C09140=1188.823,174.713,-56.680,-178.031,6.459,148.597
C09141=1188.828,174.463,-56.658,-178.034,6.458,148.598
C09142=1188.832,174.215,-56.637,-178.036,6.457,148.598
C09143=1188.837,173.966,-56.613,-178.039,6.455,148.599
C09144=1188.841,173.716,-56.591,-178.041,6.453,148.599
C09145=1188.846,173.468,-56.569,-178.044,6.451,148.599
C09146=1188.851,173.219,-56.546,-178.047,6.450,148.600
C09147=1188.856,172.970,-56.524,-178.049,6.448,148.600
C09148=1188.860,172.721,-56.502,-178.052,6.446,148.600
C09149=1188.865,172.472,-56.479,-178.055,6.444,148.601
C09150=1188.870,172.223,-56.457,-178.057,6.442,148.601
C09151=1188.874,171.974,-56.435,-178.060,6.441,148.601
C09152=1188.879,171.725,-56.412,-178.063,6.439,148.602
C09153=1188.884,171.476,-56.390,-178.065,6.437,148.602
C09154=1188.888,171.228,-56.369,-178.068,6.435,148.603
C09155=1188.893,170.978,-56.347,-178.071,6.433,148.603
C09156=1188.898,170.729,-56.324,-178.073,6.432,148.603
C09157=1188.902,170.480,-56.301,-178.076,6.430,148.604
C09158=1188.907,170.231,-56.279,-178.079,6.428,148.604
C09159=1188.911,169.983,-56.258,-178.081,6.426,148.604
C09160=1188.916,169.733,-56.235,-178.084,6.425,148.605
C09161=1188.921,169.484,-56.213,-178.087,6.423,148.605
C09162=1188.925,169.235,-56.191,-178.089,6.422,148.605
C09163=1188.930,168.987,-56.169,-178.092,6.420,148.606
C09164=1188.935,168.737,-56.146,-178.095,6.419,148.606
C09165=1188.940,168.489,-56.125,-178.097,6.417,148.607
C09166=1188.944,168.239,-56.103,-178.100,6.415,148.607
C09167=1188.949,167.991,-56.081,-178.103,6.413,148.608
C09168=1188.953,167.741,-56.059,-178.105,6.411,148.608
C09169=1188.958,167.493,-56.037,-178.108,6.410,148.608
C09170=1188.963,167.243,-56.015,-178.111,6.408,148.609
C09171=1188.968,166.994,-55.993,-178.114,6.406,148.609
C09172=1188.972,166.745,-55.971,-178.116,6.404,148.609
C09173=1188.977,166.496,-55.949,-178.119,6.403,148.610
C09174=1188.982,166.247,-55.927,-178.122,6.401,148.610
C09175=1188.986,165.998,-55.905,-178.124,6.400,148.610
C09176=1188.991,165.750,-55.884,-178.126,6.398,148.611
C09177=1188.996,165.500,-55.862,-178.129,6.396,148.611
C09178=1189.001,165.251,-55.839,-178.132,6.394,148.612
C09179=1189.005,165.002,-55.817,-178.134,6.393,148.612
C09180=1189.010,164.753,-55.796,-178.137,6.391,148.612
C09181=1189.015,164.504,-55.774,-178.140,6.389,148.613
C09182=1189.019,164.255,-55.752,-178.142,6.387,148.613
C09183=1189.024,164.006,-55.730,-178.146,6.386,148.614
C09184=1189.029,163.757,-55.708,-178.148,6.384,148.614
C09185=1189.033,163.509,-55.687,-178.151,6.382,148.614
C09186=1189.038,163.259,-55.664,-178.153,6.381,148.615
C09187=1189.043,163.011,-55.643,-178.156,6.380,148.615
C09188=1189.047,162.762,-55.621,-178.158,6.378,148.616
C09189=1189.052,162.512,-55.600,-178.161,6.376,148.616
C09190=1189.057,162.264,-55.578,-178.164,6.374,148.616
C09191=1189.061,162.014,-55.556,-178.166,6.372,148.617
C09192=1189.066,161.766,-55.534,-178.169,6.371,148.617
C09193=1189.070,161.516,-55.512,-178.172,6.369,148.617
C09194=1189.075,161.268,-55.491,-178.174,6.368,148.618
C09195=1189.080,161.018,-55.470,-178.177,6.366,148.618
C09196=1189.085,160.769,-55.448,-178.180,6.365,148.619
C09197=1189.089,160.520,-55.426,-178.182,6.363,148.619
C09198=1189.094,160.272,-55.404,-178.185,6.361,148.619
C09199=1189.099,160.022,-55.383,-178.188,6.359,148.620
C09200=1189.104,159.773,-55.361,-178.190,6.358,148.620
C09201=1189.109,159.525,-55.340,-178.193,6.356,148.621
C09202=1189.112,159.276,-55.318,-178.195,6.355,148.621
C09203=1189.118,159.006,-55.295,-178.198,6.352,148.621
C09204=1189.123,158.737,-55.271,-178.202,6.351,148.622
C09205=1189.128,158.468,-55.248,-178.204,6.349,148.622
C09206=1189.132,158.199,-55.225,-178.207,6.347,148.623
C09207=1189.138,157.950,-55.204,-178.210,6.346,148.623
C09208=1189.142,157.701,-55.182,-178.212,6.344,148.623
C09209=1189.147,157.453,-55.161,-178.215,6.343,148.624
C09210=1189.152,157.203,-55.139,-178.218,6.341,148.624
C09211=1189.157,156.954,-55.118,-178.220,6.340,148.625
C09212=1189.162,156.706,-55.096,-178.223,6.338,148.625
C09213=1189.166,156.456,-55.075,-178.226,6.336,148.626
C09214=1189.170,156.207,-55.054,-178.228,6.334,148.626
C09215=1189.175,155.958,-55.033,-178.230,6.333,148.626
C09216=1189.180,155.709,-55.011,-178.233,6.332,148.627
C09217=1189.185,155.459,-54.990,-178.236,6.330,148.627
C09218=1189.190,155.211,-54.968,-178.239,6.328,148.628
C09219=1189.194,154.962,-54.947,-178.242,6.327,148.628
C09220=1189.199,154.713,-54.926,-178.244,6.325,148.628
C09221=1189.203,154.464,-54.904,-178.247,6.323,148.629
C09222=1189.209,154.215,-54.883,-178.249,6.322,148.629
C09223=1189.213,153.966,-54.861,-178.252,6.320,148.630
C09224=1189.218,153.717,-54.841,-178.255,6.319,148.630
C09225=1189.222,153.468,-54.819,-178.258,6.317,148.631
C09226=1189.227,153.218,-54.798,-178.260,6.315,148.631
C09227=1189.232,152.969,-54.777,-178.262,6.314,148.631
C09228=1189.237,152.721,-54.756,-178.265,6.313,148.632
C09229=1189.241,152.471,-54.734,-178.268,6.311,148.632
C09230=1189.246,152.222,-54.713,-178.271,6.309,148.632
C09231=1189.250,151.973,-54.692,-178.273,6.307,148.633
C09232=1189.256,151.724,-54.671,-178.276,6.306,148.633
C09233=1189.260,151.475,-54.650,-178.278,6.305,148.634
C09234=1189.266,151.226,-54.629,-178.281,6.303,148.634
C09235=1189.269,150.977,-54.607,-178.284,6.301,148.635
C09236=1189.274,150.728,-54.586,-178.287,6.300,148.635
C09237=1189.280,150.478,-54.565,-178.289,6.298,148.635
C09238=1189.284,150.230,-54.544,-178.292,6.297,148.636
C09239=1189.289,149.981,-54.523,-178.294,6.295,148.636
C09240=1189.293,149.732,-54.503,-178.297,6.294,148.637
C09241=1189.298,149.483,-54.481,-178.300,6.292,148.637
C09242=1189.303,149.233,-54.460,-178.303,6.290,148.637
C09243=1189.307,148.984,-54.440,-178.305,6.289,148.638
C09244=1189.312,148.735,-54.419,-178.308,6.288,148.638
C09245=1189.317,148.487,-54.397,-178.311,6.286,148.639
C09246=1189.322,148.238,-54.377,-178.313,6.284,148.639
C09247=1189.327,147.988,-54.356,-178.316,6.282,148.640
C09248=1189.331,147.739,-54.335,-178.318,6.281,148.640
C09249=1189.336,147.490,-54.313,-178.321,6.280,148.640
C09250=1189.341,147.241,-54.292,-178.324,6.278,148.641
C09251=1189.345,146.992,-54.272,-178.327,6.277,148.641
C09252=1189.350,146.743,-54.251,-178.329,6.275,148.642
C09253=1189.355,146.494,-54.231,-178.331,6.274,148.642
C09254=1189.360,146.245,-54.209,-178.334,6.272,148.643
C09255=1189.364,145.996,-54.188,-178.337,6.270,148.643
C09256=1189.369,145.747,-54.168,-178.340,6.269,148.643
C09257=1189.373,145.497,-54.147,-178.342,6.268,148.644
C09258=1189.378,145.248,-54.126,-178.345,6.266,148.644
C09259=1189.383,144.999,-54.105,-178.347,6.264,148.645
C09260=1189.388,144.750,-54.084,-178.350,6.263,148.645
C09261=1189.392,144.501,-54.064,-178.353,6.261,148.646
C09262=1189.397,144.251,-54.043,-178.355,6.260,148.646
C09263=1189.402,144.003,-54.022,-178.358,6.258,148.646
C09264=1189.407,143.754,-54.001,-178.361,6.257,148.647
C09265=1189.411,143.505,-53.981,-178.363,6.255,148.647
C09266=1189.416,143.256,-53.960,-178.366,6.254,148.648
C09267=1189.421,143.007,-53.939,-178.369,6.253,148.648
C09268=1189.426,142.757,-53.918,-178.371,6.251,148.649
C09269=1189.430,142.508,-53.898,-178.374,6.249,148.649
C09270=1189.435,142.260,-53.878,-178.376,6.248,148.649
C09271=1189.440,142.010,-53.857,-178.379,6.247,148.650
C09272=1189.444,141.761,-53.836,-178.382,6.245,148.650
C09273=1189.450,141.512,-53.815,-178.385,6.243,148.651
C09274=1189.454,141.263,-53.795,-178.387,6.242,148.651
C09275=1189.459,141.014,-53.775,-178.390,6.241,148.652
C09276=1189.464,140.764,-53.754,-178.393,6.239,148.652
C09277=1189.468,140.515,-53.734,-178.395,6.237,148.653
C09278=1189.474,140.266,-53.713,-178.398,6.236,148.653
C09279=1189.478,140.017,-53.693,-178.400,6.235,148.653
C09280=1189.482,139.768,-53.672,-178.403,6.233,148.654
C09281=1189.488,139.519,-53.651,-178.405,6.232,148.654
C09282=1189.492,139.270,-53.631,-178.408,6.230,148.655
C09283=1189.497,139.021,-53.611,-178.411,6.229,148.655
C09284=1189.502,138.772,-53.590,-178.414,6.227,148.656
C09285=1189.506,138.522,-53.570,-178.416,6.226,148.656
C09286=1189.511,138.273,-53.550,-178.419,6.225,148.656
C09287=1189.516,138.024,-53.529,-178.422,6.223,148.657
C09288=1189.521,137.775,-53.508,-178.425,6.221,148.657
C09289=1189.525,137.526,-53.488,-178.427,6.220,148.658
C09290=1189.530,137.277,-53.468,-178.430,6.219,148.658
C09291=1189.535,137.027,-53.447,-178.432,6.217,148.659
C09292=1189.539,136.778,-53.427,-178.434,6.216,148.659
C09293=1189.544,136.529,-53.406,-178.438,6.215,148.660
C09294=1189.548,136.280,-53.386,-178.440,6.213,148.660
C09295=1189.554,136.031,-53.366,-178.443,6.211,148.660
C09296=1189.559,135.782,-53.346,-178.445,6.210,148.661
C09297=1189.563,135.533,-53.325,-178.448,6.209,148.661
C09298=1189.568,135.284,-53.306,-178.451,6.207,148.662
C09299=1189.573,135.034,-53.285,-178.453,6.206,148.662
C09300=1189.577,134.786,-53.264,-178.456,6.204,148.663
C09301=1189.582,134.536,-53.245,-178.459,6.203,148.663
C09302=1189.587,134.287,-53.224,-178.462,6.201,148.664
C09303=1189.592,134.038,-53.203,-178.464,6.200,148.664
C09304=1189.597,133.788,-53.184,-178.467,6.199,148.665
C09305=1189.602,133.540,-53.164,-178.470,6.197,148.665
C09306=1189.606,133.291,-53.143,-178.472,6.196,148.665
C09307=1189.612,133.022,-53.122,-178.475,6.195,148.666
C09308=1189.616,132.754,-53.100,-178.478,6.193,148.666
C09309=1189.622,132.485,-53.078,-178.480,6.191,148.667
C09310=1189.627,132.216,-53.057,-178.483,6.190,148.667
C09311=1189.631,131.967,-53.037,-178.486,6.188,148.668
C09312=1189.636,131.718,-53.017,-178.488,6.187,148.668
C09313=1189.641,131.469,-52.996,-178.491,6.186,148.669
C09314=1189.646,131.219,-52.977,-178.494,6.184,148.669
C09315=1189.650,130.970,-52.956,-178.496,6.183,148.670
C09316=1189.655,130.722,-52.936,-178.499,6.181,148.670
C09317=1189.660,130.472,-52.917,-178.502,6.180,148.671
C09318=1189.665,130.223,-52.896,-178.504,6.179,148.671
C09319=1189.669,129.974,-52.876,-178.507,6.177,148.671
C09320=1189.674,129.724,-52.857,-178.510,6.176,148.672
C09321=1189.679,129.476,-52.837,-178.512,6.175,148.672
C09322=1189.684,129.226,-52.817,-178.515,6.173,148.673
C09323=1189.688,128.977,-52.797,-178.518,6.171,148.673
C09324=1189.693,128.728,-52.777,-178.520,6.171,148.674
C09325=1189.698,128.479,-52.756,-178.523,6.169,148.674
C09326=1189.704,128.230,-52.737,-178.526,6.167,148.675
C09327=1189.708,127.981,-52.717,-178.528,6.166,148.675
C09328=1189.713,127.731,-52.697,-178.531,6.165,148.676
C09329=1189.718,127.482,-52.677,-178.534,6.163,148.676
C09330=1189.723,127.233,-52.657,-178.536,6.162,148.677
C09331=1189.727,126.984,-52.638,-178.539,6.161,148.677
C09332=1189.732,126.734,-52.618,-178.542,6.159,148.678
C09333=1189.736,126.485,-52.598,-178.544,6.158,148.678
C09334=1189.742,126.236,-52.578,-178.547,6.156,148.679
C09335=1189.746,125.987,-52.559,-178.550,6.155,148.679
C09336=1189.750,125.738,-52.539,-178.552,6.154,148.679
C09337=1189.755,125.489,-52.519,-178.555,6.152,148.680
C09338=1189.760,125.240,-52.500,-178.557,6.151,148.680
C09339=1189.765,124.991,-52.479,-178.560,6.150,148.681
C09340=1189.770,124.741,-52.460,-178.563,6.148,148.681
C09341=1189.775,124.492,-52.441,-178.565,6.147,148.682
C09342=1189.780,124.243,-52.421,-178.568,6.146,148.682
C09343=1189.784,123.994,-52.401,-178.571,6.144,148.683
C09344=1189.789,123.744,-52.381,-178.573,6.143,148.683
C09345=1189.794,123.495,-52.362,-178.576,6.141,148.684
C09346=1189.799,123.246,-52.342,-178.578,6.141,148.684
C09347=1189.803,122.997,-52.322,-178.581,6.139,148.685
C09348=1189.808,122.748,-52.303,-178.584,6.137,148.685
C09349=1189.813,122.499,-52.283,-178.586,6.137,148.686
C09350=1189.817,122.249,-52.264,-178.589,6.135,148.686
C09351=1189.823,122.000,-52.244,-178.592,6.133,148.686
C09352=1189.828,121.751,-52.225,-178.594,6.133,148.687
C09353=1189.832,121.502,-52.204,-178.597,6.131,148.687
C09354=1189.837,121.253,-52.185,-178.599,6.130,148.688
C09355=1189.841,121.004,-52.166,-178.602,6.129,148.689
C09356=1189.846,120.754,-52.146,-178.605,6.127,148.689
C09357=1189.851,120.505,-52.127,-178.607,6.126,148.689
C09358=1189.856,120.256,-52.107,-178.610,6.125,148.690
C09359=1189.861,120.007,-52.088,-178.612,6.124,148.690
C09360=1189.865,119.758,-52.069,-178.615,6.122,148.691
C09361=1189.870,119.508,-52.049,-178.618,6.120,148.691
C09362=1189.876,119.259,-52.030,-178.620,6.120,148.692
C09363=1189.880,119.010,-52.010,-178.623,6.118,148.692
C09364=1189.885,118.761,-51.990,-178.626,6.117,148.693
C09365=1189.889,118.512,-51.971,-178.628,6.115,148.693
C09366=1189.894,118.263,-51.952,-178.631,6.114,148.694
C09367=1189.899,118.014,-51.932,-178.634,6.113,148.694
C09368=1189.904,117.764,-51.913,-178.636,6.111,148.695
C09369=1189.909,117.516,-51.894,-178.639,6.110,148.695
C09370=1189.914,117.265,-51.875,-178.642,6.109,148.696
C09371=1189.919,117.016,-51.855,-178.644,6.107,148.696
C09372=1189.924,116.767,-51.836,-178.647,6.107,148.697
C09373=1189.928,116.518,-51.817,-178.650,6.105,148.697
C09374=1189.933,116.269,-51.798,-178.652,6.104,148.698
C09375=1189.938,116.019,-51.778,-178.655,6.103,148.698
C09376=1189.943,115.771,-51.759,-178.658,6.101,148.699
C09377=1189.947,115.521,-51.740,-178.660,6.100,148.699
C09378=1189.952,115.272,-51.720,-178.663,6.099,148.700
C09379=1189.957,115.023,-51.701,-178.665,6.098,148.700
C09380=1189.961,114.773,-51.682,-178.668,6.096,148.700
C09381=1189.967,114.525,-51.662,-178.671,6.095,148.701
C09382=1189.971,114.275,-51.644,-178.673,6.094,148.701
C09383=1189.976,114.026,-51.625,-178.676,6.092,148.702
C09384=1189.981,113.776,-51.605,-178.679,6.091,148.703
C09385=1189.986,113.528,-51.586,-178.681,6.090,148.703
C09386=1189.991,113.278,-51.567,-178.684,6.089,148.704
C09387=1189.995,113.029,-51.549,-178.687,6.087,148.704
C09388=1190.000,112.779,-51.529,-178.689,6.087,148.705
C09389=1190.006,112.531,-51.510,-178.692,6.085,148.705
C09390=1190.010,112.281,-51.491,-178.694,6.084,148.705
C09391=1190.015,112.032,-51.471,-178.697,6.083,148.706
C09392=1190.019,111.783,-51.453,-178.700,6.081,148.706
C09393=1190.025,111.534,-51.434,-178.702,6.080,148.707
C09394=1190.029,111.284,-51.414,-178.705,6.078,148.707
C09395=1190.034,111.036,-51.395,-178.707,6.078,148.708
C09396=1190.039,110.785,-51.377,-178.711,6.076,148.709
C09397=1190.044,110.537,-51.358,-178.713,6.075,148.709
C09398=1190.049,110.288,-51.339,-178.715,6.074,148.709
C09399=1190.053,110.038,-51.320,-178.718,6.073,148.710
C09400=1190.059,109.789,-51.301,-178.721,6.071,148.710
C09401=1190.063,109.540,-51.282,-178.723,6.071,148.711
C09402=1190.068,109.290,-51.263,-178.726,6.069,148.711
C09403=1190.072,109.041,-51.244,-178.729,6.067,148.712
C09404=1190.078,108.792,-51.225,-178.731,6.067,148.712
C09405=1190.082,108.542,-51.207,-178.734,6.065,148.713
C09406=1190.087,108.294,-51.187,-178.737,6.064,148.714
C09407=1190.092,108.044,-51.169,-178.739,6.062,148.714
C09408=1190.097,107.795,-51.150,-178.742,6.062,148.714
C09409=1190.101,107.546,-51.131,-178.745,6.060,148.715
C09410=1190.107,107.296,-51.112,-178.747,6.059,148.715
C09411=1190.111,107.028,-51.092,-178.750,6.058,148.716
C09412=1190.117,106.760,-51.072,-178.753,6.056,148.716
C09413=1190.122,106.491,-51.051,-178.755,6.056,148.717
C09414=1190.127,106.223,-51.031,-178.759,6.054,148.718
C09415=1190.132,105.974,-51.012,-178.761,6.052,148.718
C09416=1190.137,105.724,-50.994,-178.764,6.052,148.719
C09417=1190.141,105.476,-50.975,-178.767,6.050,148.719
C09418=1190.147,105.226,-50.956,-178.769,6.049,148.720
C09419=1190.151,104.977,-50.937,-178.772,6.048,148.720
C09420=1190.157,104.727,-50.919,-178.774,6.047,148.721
C09421=1190.161,104.478,-50.900,-178.777,6.046,148.721
C09422=1190.166,104.229,-50.882,-178.779,6.045,148.722
C09423=1190.171,103.980,-50.863,-178.782,6.043,148.722
C09424=1190.175,103.730,-50.844,-178.785,6.042,148.723
C09425=1190.180,103.481,-50.826,-178.787,6.041,148.723
C09426=1190.186,103.232,-50.807,-178.790,6.040,148.724
C09427=1190.190,102.982,-50.789,-178.793,6.038,148.724
C09428=1190.195,102.733,-50.770,-178.795,6.038,148.725
C09429=1190.200,102.484,-50.751,-178.798,6.036,148.725
C09430=1190.204,102.234,-50.733,-178.801,6.035,148.726
C09431=1190.209,101.986,-50.714,-178.803,6.034,148.726
C09432=1190.215,101.736,-50.696,-178.805,6.033,148.727
C09433=1190.220,101.487,-50.678,-178.809,6.031,148.727
C09434=1190.224,101.238,-50.659,-178.811,6.030,148.728
C09435=1190.229,100.988,-50.640,-178.814,6.029,148.728
C09436=1190.234,100.739,-50.622,-178.816,6.028,148.729
C09437=1190.238,100.490,-50.603,-178.819,6.027,148.729
C09438=1190.243,100.241,-50.585,-178.821,6.026,148.730
C09439=1190.249,99.991,-50.566,-178.825,6.024,148.731
C09440=1190.254,99.742,-50.548,-178.827,6.023,148.731
C09441=1190.258,99.493,-50.529,-178.829,6.023,148.731
C09442=1190.263,99.244,-50.511,-178.832,6.021,148.732
C09443=1190.268,98.994,-50.493,-178.834,6.020,148.732
C09444=1190.272,98.745,-50.474,-178.837,6.019,148.733
C09445=1190.277,98.496,-50.456,-178.840,6.018,148.733
C09446=1190.282,98.247,-50.438,-178.843,6.017,148.734
C09447=1190.288,97.997,-50.419,-178.845,6.016,148.735
C09448=1190.292,97.747,-50.401,-178.848,6.014,148.735
C09449=1190.297,97.499,-50.382,-178.850,6.013,148.736
C09450=1190.301,97.250,-50.364,-178.853,6.012,148.736
C09451=1190.306,97.000,-50.346,-178.856,6.011,148.737
C09452=1190.312,96.751,-50.328,-178.859,6.010,148.737
C09453=1190.316,96.501,-50.309,-178.861,6.009,148.738
C09454=1190.321,96.252,-50.291,-178.864,6.007,148.738
C09455=1190.326,96.003,-50.273,-178.866,6.006,148.739
C09456=1190.331,95.754,-50.255,-178.868,6.006,148.739
C09457=1190.336,95.505,-50.237,-178.872,6.004,148.740
C09458=1190.340,95.255,-50.218,-178.874,6.003,148.740
C09459=1190.346,95.006,-50.200,-178.877,6.002,148.741
C09460=1190.351,94.756,-50.182,-178.879,6.001,148.741
C09461=1190.355,94.507,-50.164,-178.882,6.000,148.742
C09462=1190.360,94.258,-50.146,-178.884,5.999,148.742
C09463=1190.365,94.008,-50.128,-178.888,5.997,148.743
C09464=1190.370,93.759,-50.110,-178.890,5.996,148.743
C09465=1190.375,93.510,-50.092,-178.892,5.996,148.744
C09466=1190.379,93.261,-50.074,-178.895,5.994,148.744
C09467=1190.384,93.011,-50.056,-178.898,5.994,148.745
C09468=1190.389,92.762,-50.038,-178.900,5.992,148.746
C09469=1190.394,92.512,-50.019,-178.903,5.991,148.746
C09470=1190.399,92.263,-50.001,-178.906,5.990,148.747
C09471=1190.404,92.014,-49.983,-178.908,5.989,148.747
C09472=1190.409,91.765,-49.965,-178.910,5.988,148.748
C09473=1190.414,91.515,-49.947,-178.914,5.987,148.748
C09474=1190.419,91.266,-49.929,-178.916,5.986,148.749
C09475=1190.424,91.017,-49.911,-178.919,5.984,148.749
C09476=1190.429,90.768,-49.893,-178.921,5.983,148.750
C09477=1190.433,90.518,-49.874,-178.924,5.982,148.750
C09478=1190.438,90.269,-49.856,-178.926,5.981,148.751
C09479=1190.443,90.020,-49.838,-178.929,5.981,148.752
C09480=1190.448,89.770,-49.821,-178.932,5.979,148.752
C09481=1190.453,89.521,-49.803,-178.934,5.978,148.753
C09482=1190.458,89.272,-49.785,-178.937,5.977,148.753
C09483=1190.463,89.022,-49.767,-178.940,5.976,148.754
C09484=1190.468,88.773,-49.749,-178.942,5.975,148.754
C09485=1190.473,88.524,-49.731,-178.945,5.974,148.755
C09486=1190.478,88.275,-49.713,-178.947,5.973,148.755
C09487=1190.481,88.025,-49.696,-178.950,5.971,148.756
C09488=1190.486,87.776,-49.678,-178.953,5.971,148.756
C09489=1190.491,87.526,-49.660,-178.955,5.970,148.757
C09490=1190.496,87.277,-49.642,-178.958,5.968,148.757
C09491=1190.501,87.028,-49.624,-178.960,5.968,148.758
C09492=1190.506,86.779,-49.606,-178.963,5.966,148.758
C09493=1190.511,86.530,-49.588,-178.966,5.965,148.759
C09494=1190.516,86.280,-49.571,-178.968,5.965,148.759
C09495=1190.521,86.031,-49.553,-178.971,5.963,148.760
C09496=1190.526,85.781,-49.535,-178.973,5.962,148.761
C09497=1190.531,85.532,-49.517,-178.976,5.961,148.761
C09498=1190.535,85.283,-49.501,-178.979,5.960,148.762
C09499=1190.540,85.034,-49.483,-178.981,5.959,148.762
C09500=1190.545,84.784,-49.465,-178.984,5.958,148.763
C09501=1190.550,84.535,-49.447,-178.987,5.957,148.763
C09502=1190.555,84.285,-49.429,-178.989,5.955,148.764
C09503=1190.560,84.036,-49.411,-178.992,5.955,148.764
C09504=1190.565,83.787,-49.395,-178.994,5.954,148.765
C09505=1190.570,83.538,-49.377,-178.997,5.953,148.765
C09506=1190.574,83.288,-49.359,-178.999,5.952,148.766
C09507=1190.580,83.039,-49.341,-179.002,5.951,148.767
C09508=1190.585,82.789,-49.324,-179.005,5.950,148.767
C09509=1190.590,82.540,-49.306,-179.007,5.949,148.768
C09510=1190.594,82.291,-49.289,-179.011,5.947,148.768
C09511=1190.599,82.042,-49.271,-179.013,5.947,148.769
C09512=1190.604,81.792,-49.253,-179.015,5.946,148.769
C09513=1190.609,81.543,-49.236,-179.018,5.944,148.770
C09514=1190.613,81.294,-49.218,-179.021,5.944,148.770
C09515=1190.619,81.025,-49.200,-179.024,5.942,148.771
C09516=1190.624,80.757,-49.181,-179.026,5.941,148.771
C09517=1190.630,80.488,-49.162,-179.029,5.940,148.772
C09518=1190.635,80.220,-49.143,-179.032,5.940,148.773
C09519=1190.639,79.971,-49.126,-179.034,5.939,148.773
C09520=1190.644,79.721,-49.108,-179.037,5.937,148.774
C09521=1190.649,79.472,-49.090,-179.039,5.936,148.774
C09522=1190.655,79.222,-49.073,-179.043,5.935,148.775
C09523=1190.659,78.973,-49.056,-179.045,5.934,148.775
C09524=1190.664,78.723,-49.039,-179.047,5.934,148.776
C09525=1190.669,78.475,-49.021,-179.051,5.932,148.777
C09526=1190.674,78.225,-49.004,-179.053,5.931,148.777
C09527=1190.679,77.976,-48.986,-179.055,5.931,148.778
C09528=1190.684,77.726,-48.969,-179.058,5.929,148.778
C09529=1190.688,77.478,-48.952,-179.061,5.928,148.779
C09530=1190.693,77.228,-48.934,-179.063,5.928,148.779
C09531=1190.698,76.979,-48.916,-179.066,5.926,148.780
C09532=1190.703,76.729,-48.900,-179.068,5.925,148.780
C09533=1190.708,76.479,-48.882,-179.071,5.925,148.781
C09534=1190.714,76.231,-48.865,-179.074,5.923,148.782
C09535=1190.718,75.981,-48.848,-179.076,5.922,148.782
C09536=1190.723,75.732,-48.831,-179.079,5.922,148.783
C09537=1190.728,75.482,-48.813,-179.081,5.920,148.783
C09538=1190.733,75.233,-48.796,-179.084,5.920,148.784
C09539=1190.738,74.983,-48.779,-179.086,5.919,148.784
C09540=1190.742,74.734,-48.762,-179.089,5.917,148.785
C09541=1190.748,74.485,-48.745,-179.092,5.917,148.786
C09542=1190.753,74.235,-48.727,-179.094,5.916,148.786
C09543=1190.757,73.986,-48.710,-179.097,5.915,148.787
C09544=1190.763,73.737,-48.693,-179.100,5.914,148.787
C09545=1190.767,73.487,-48.676,-179.102,5.913,148.788
C09546=1190.772,73.238,-48.658,-179.104,5.912,148.788
C09547=1190.777,72.989,-48.642,-179.108,5.911,148.789
C09548=1190.782,72.739,-48.625,-179.110,5.910,148.789
C09549=1190.787,72.490,-48.608,-179.112,5.909,148.790
C09550=1190.792,72.241,-48.590,-179.116,5.908,148.791
C09551=1190.797,71.991,-48.573,-179.118,5.907,148.791
C09552=1190.802,71.742,-48.556,-179.120,5.907,148.792
C09553=1190.807,71.492,-48.539,-179.123,5.905,148.792
C09554=1190.812,71.243,-48.522,-179.126,5.904,148.793
C09555=1190.817,70.994,-48.504,-179.128,5.904,148.793
C09556=1190.821,70.744,-48.488,-179.131,5.902,148.794
C09557=1190.827,70.495,-48.471,-179.134,5.902,148.794
C09558=1190.831,70.246,-48.454,-179.136,5.901,148.795
C09559=1190.836,69.996,-48.438,-179.138,5.900,148.796
C09560=1190.841,69.746,-48.420,-179.142,5.899,148.796
C09561=1190.846,69.498,-48.403,-179.144,5.898,148.797
C09562=1190.851,69.248,-48.386,-179.146,5.897,148.797
C09563=1190.855,68.999,-48.369,-179.149,5.896,148.798
C09564=1190.861,68.749,-48.352,-179.152,5.895,148.798
C09565=1190.866,68.500,-48.336,-179.154,5.894,148.799
C09566=1190.871,68.251,-48.319,-179.156,5.894,148.800
C09567=1190.875,68.001,-48.302,-179.160,5.892,148.800
C09568=1190.880,67.752,-48.285,-179.162,5.891,148.801
C09569=1190.886,67.503,-48.268,-179.164,5.891,148.801
C09570=1190.890,67.253,-48.252,-179.167,5.889,148.802
C09571=1190.895,67.003,-48.234,-179.170,5.889,148.802
C09572=1190.900,66.754,-48.217,-179.172,5.888,148.803
C09573=1190.905,66.506,-48.201,-179.175,5.887,148.803
C09574=1190.910,66.256,-48.183,-179.178,5.886,148.804
C09575=1190.914,66.006,-48.167,-179.180,5.885,148.805
C09576=1190.919,65.758,-48.150,-179.183,5.884,148.805
C09577=1190.925,65.508,-48.133,-179.186,5.883,148.806
C09578=1190.929,65.258,-48.117,-179.188,5.882,148.806
C09579=1190.934,65.008,-48.099,-179.191,5.882,148.807
C09580=1190.940,64.759,-48.084,-179.193,5.881,148.808
C09581=1190.944,64.510,-48.067,-179.196,5.879,148.808
C09582=1190.949,64.260,-48.050,-179.199,5.879,148.809
C09583=1190.955,64.011,-48.033,-179.201,5.878,148.809
C09584=1190.959,63.761,-48.017,-179.203,5.877,148.810
C09585=1190.964,63.512,-48.000,-179.207,5.876,148.810
C09586=1190.969,63.263,-47.983,-179.209,5.875,148.811
C09587=1190.974,63.013,-47.967,-179.211,5.875,148.812
C09588=1190.978,62.764,-47.950,-179.213,5.874,148.812
C09589=1190.984,62.515,-47.933,-179.217,5.872,148.813
C09590=1190.989,62.265,-47.916,-179.219,5.872,148.813
C09591=1190.994,62.016,-47.901,-179.221,5.871,148.814
C09592=1190.998,61.766,-47.884,-179.224,5.870,148.814
C09593=1191.004,61.517,-47.867,-179.227,5.869,148.815
C09594=1191.009,61.268,-47.850,-179.229,5.868,148.816
C09595=1191.013,61.018,-47.834,-179.232,5.868,148.816
C09596=1191.018,60.769,-47.817,-179.234,5.867,148.817
C09597=1191.024,60.519,-47.801,-179.237,5.865,148.817
C09598=1191.028,60.270,-47.784,-179.240,5.865,148.818
C09599=1191.033,60.021,-47.768,-179.242,5.864,148.818
C09600=1191.038,59.771,-47.751,-179.245,5.863,148.819
C09601=1191.043,59.522,-47.734,-179.248,5.862,148.819
C09602=1191.049,59.272,-47.718,-179.250,5.861,148.820
C09603=1191.053,59.023,-47.702,-179.253,5.861,148.821
C09604=1191.058,58.774,-47.685,-179.255,5.860,148.821
C09605=1191.063,58.525,-47.669,-179.258,5.859,148.822
C09606=1191.069,58.275,-47.653,-179.261,5.858,148.823
C09607=1191.073,58.025,-47.636,-179.263,5.857,148.823
C09608=1191.078,57.776,-47.619,-179.266,5.856,148.824
C09609=1191.083,57.526,-47.604,-179.268,5.856,148.824
C09610=1191.088,57.277,-47.587,-179.271,5.854,148.825
C09611=1191.093,57.028,-47.571,-179.274,5.854,148.825
C09612=1191.097,56.778,-47.555,-179.276,5.853,148.826
C09613=1191.103,56.529,-47.538,-179.278,5.852,148.827
C09614=1191.108,56.279,-47.521,-179.281,5.852,148.827
C09615=1191.113,56.030,-47.506,-179.284,5.850,148.828
C09616=1191.118,55.781,-47.489,-179.286,5.850,148.828
C09617=1191.122,55.531,-47.472,-179.289,5.849,148.829
C09618=1191.127,55.282,-47.457,-179.291,5.848,148.829
C09619=1191.133,55.014,-47.439,-179.294,5.847,148.830
C09620=1191.138,54.745,-47.422,-179.297,5.846,148.831
C09621=1191.144,54.476,-47.404,-179.300,5.846,148.831
C09622=1191.149,54.208,-47.386,-179.303,5.844,148.832
C09623=1191.154,53.958,-47.370,-179.305,5.843,148.833
C09624=1191.159,53.709,-47.354,-179.308,5.843,148.833
C09625=1191.164,53.460,-47.337,-179.310,5.842,148.834
C09626=1191.169,53.210,-47.322,-179.313,5.841,148.834
C09627=1191.173,52.961,-47.305,-179.316,5.840,148.835
C09628=1191.179,52.711,-47.289,-179.318,5.840,148.836
C09629=1191.183,52.462,-47.273,-179.321,5.839,148.836
C09630=1191.189,52.212,-47.257,-179.323,5.838,148.837
C09631=1191.193,51.963,-47.241,-179.326,5.837,148.837
C09632=1191.198,51.714,-47.225,-179.329,5.836,148.838
C09633=1191.203,51.464,-47.208,-179.331,5.835,148.839
C09634=1191.208,51.215,-47.193,-179.333,5.835,148.839
C09635=1191.213,50.965,-47.176,-179.336,5.834,148.840
C09636=1191.218,50.716,-47.160,-179.339,5.834,148.840
C09637=1191.223,50.466,-47.144,-179.341,5.832,148.841
C09638=1191.228,50.217,-47.128,-179.344,5.831,148.841
C09639=1191.233,49.968,-47.113,-179.347,5.831,148.842
C09640=1191.238,49.718,-47.096,-179.349,5.830,148.842
C09641=1191.243,49.469,-47.080,-179.351,5.829,148.843
C09642=1191.248,49.219,-47.064,-179.355,5.828,148.844
C09643=1191.253,48.970,-47.048,-179.357,5.827,148.844
C09644=1191.258,48.720,-47.032,-179.359,5.827,148.845
C09645=1191.263,48.471,-47.016,-179.362,5.826,148.846
C09646=1191.268,48.221,-47.000,-179.364,5.825,148.846
C09647=1191.273,47.971,-46.984,-179.367,5.825,148.847
C09648=1191.278,47.723,-46.969,-179.370,5.823,148.847
C09649=1191.282,47.473,-46.953,-179.372,5.822,148.848
C09650=1191.288,47.223,-46.937,-179.375,5.822,148.849
C09651=1191.293,46.975,-46.921,-179.377,5.821,148.849
C09652=1191.298,46.724,-46.905,-179.380,5.821,148.850
C09653=1191.303,46.475,-46.889,-179.382,5.820,148.850
C09654=1191.308,46.226,-46.872,-179.385,5.819,148.851
C09655=1191.313,45.976,-46.857,-179.388,5.818,148.851
C09656=1191.318,45.727,-46.841,-179.390,5.817,148.852
C09657=1191.322,45.478,-46.825,-179.393,5.817,148.853
C09658=1191.327,45.228,-46.810,-179.395,5.816,148.853
C09659=1191.333,44.979,-46.794,-179.398,5.815,148.854
C09660=1191.338,44.729,-46.778,-179.400,5.815,148.855
C09661=1191.343,44.480,-46.762,-179.404,5.814,148.855
C09662=1191.348,44.231,-46.746,-179.406,5.813,148.856
C09663=1191.352,43.981,-46.731,-179.408,5.812,148.856
C09664=1191.357,43.731,-46.715,-179.411,5.812,148.857
C09665=1191.363,43.482,-46.700,-179.413,5.811,148.857
C09666=1191.367,43.232,-46.683,-179.416,5.810,148.858
C09667=1191.373,42.983,-46.667,-179.419,5.809,148.859
C09668=1191.377,42.734,-46.652,-179.421,5.808,148.859
C09669=1191.382,42.484,-46.636,-179.424,5.807,148.860
C09670=1191.388,42.234,-46.621,-179.426,5.807,148.861
C09671=1191.393,41.985,-46.605,-179.429,5.806,148.861
C09672=1191.397,41.736,-46.589,-179.431,5.806,148.862
C09673=1191.402,41.486,-46.574,-179.434,5.805,148.862
C09674=1191.407,41.237,-46.558,-179.436,5.804,148.863
C09675=1191.412,40.987,-46.542,-179.439,5.803,148.863
C09676=1191.418,40.738,-46.527,-179.442,5.802,148.864
C09677=1191.422,40.488,-46.512,-179.444,5.801,148.865
C09678=1191.428,40.239,-46.496,-179.447,5.801,148.865
C09679=1191.432,39.989,-46.480,-179.449,5.800,148.866
C09680=1191.437,39.740,-46.465,-179.452,5.800,148.867
C09681=1191.442,39.490,-46.449,-179.454,5.799,148.867
C09682=1191.448,39.241,-46.434,-179.457,5.798,148.868
C09683=1191.453,38.991,-46.418,-179.460,5.797,148.868
C09684=1191.457,38.743,-46.402,-179.462,5.796,148.869
C09685=1191.462,38.493,-46.387,-179.465,5.796,148.870
C09686=1191.468,38.244,-46.371,-179.467,5.795,148.870
C09687=1191.472,37.994,-46.356,-179.470,5.794,148.871
C09688=1191.477,37.745,-46.340,-179.472,5.794,148.871
C09689=1191.483,37.495,-46.324,-179.475,5.793,148.872
C09690=1191.487,37.246,-46.309,-179.477,5.792,148.872
C09691=1191.492,36.995,-46.294,-179.480,5.792,148.873
C09692=1191.498,36.746,-46.279,-179.483,5.791,148.874
C09693=1191.502,36.497,-46.264,-179.486,5.790,148.874
C09694=1191.508,36.247,-46.248,-179.488,5.789,148.875
C09695=1191.513,35.997,-46.232,-179.490,5.789,148.876
C09696=1191.517,35.748,-46.217,-179.493,5.788,148.876
C09697=1191.523,35.499,-46.202,-179.495,5.787,148.877
C09698=1191.527,35.250,-46.187,-179.498,5.787,148.877
C09699=1191.533,35.000,-46.171,-179.500,5.786,148.878
C09700=1191.537,34.750,-46.155,-179.503,5.786,148.879
C09701=1191.542,34.501,-46.140,-179.505,5.785,148.879
C09702=1191.547,34.252,-46.124,-179.508,5.784,148.880
C09703=1191.552,34.002,-46.110,-179.511,5.783,148.881
C09704=1191.558,33.753,-46.095,-179.513,5.782,148.881
C09705=1191.563,33.503,-46.079,-179.516,5.782,148.882
C09706=1191.567,33.253,-46.064,-179.519,5.781,148.882
C09707=1191.573,33.004,-46.048,-179.521,5.780,148.883
C09708=1191.577,32.755,-46.033,-179.523,5.780,148.883
C09709=1191.583,32.506,-46.017,-179.526,5.779,148.884
C09710=1191.588,32.256,-46.003,-179.529,5.779,148.885
C09711=1191.593,32.006,-45.988,-179.531,5.778,148.885
C09712=1191.597,31.757,-45.972,-179.533,5.777,148.886
C09713=1191.602,31.507,-45.957,-179.537,5.776,148.887
C09714=1191.607,31.257,-45.942,-179.539,5.775,148.887
C09715=1191.613,31.008,-45.927,-179.541,5.775,148.888
C09716=1191.617,30.759,-45.912,-179.544,5.774,148.888
C09717=1191.623,30.510,-45.896,-179.547,5.774,148.889
C09718=1191.628,30.260,-45.882,-179.549,5.773,148.890
C09719=1191.633,30.010,-45.866,-179.552,5.772,148.890
C09720=1191.637,29.761,-45.851,-179.554,5.772,148.891
C09721=1191.643,29.511,-45.835,-179.556,5.771,148.891
C09722=1191.648,29.262,-45.821,-179.559,5.770,148.892
C09723=1191.653,28.993,-45.804,-179.562,5.770,148.893
C09724=1191.658,28.724,-45.788,-179.565,5.769,148.893
C09725=1191.664,28.455,-45.772,-179.567,5.768,148.894
C09726=1191.669,28.187,-45.756,-179.570,5.768,148.895
C09727=1191.675,27.937,-45.741,-179.573,5.767,148.895
C09728=1191.679,27.688,-45.726,-179.575,5.766,148.896
C09729=1191.685,27.439,-45.710,-179.578,5.766,148.897
C09730=1191.690,27.189,-45.696,-179.580,5.765,148.897
C09731=1191.694,26.940,-45.681,-179.583,5.765,148.898
C09732=1191.700,26.690,-45.666,-179.585,5.764,148.898
C09733=1191.705,26.441,-45.651,-179.588,5.763,148.899
C09734=1191.710,26.191,-45.635,-179.591,5.762,148.900
C09735=1191.714,25.941,-45.621,-179.593,5.761,148.900
C09736=1191.719,25.692,-45.606,-179.596,5.761,148.901
C09737=1191.725,25.442,-45.591,-179.598,5.760,148.901
C09738=1191.729,25.193,-45.576,-179.601,5.760,148.902
C09739=1191.734,24.943,-45.562,-179.603,5.759,148.903
C09740=1191.740,24.693,-45.546,-179.606,5.758,148.903
C09741=1191.744,24.444,-45.531,-179.608,5.758,148.904
C09742=1191.749,24.195,-45.517,-179.611,5.757,148.905
C09743=1191.755,23.945,-45.501,-179.613,5.756,148.905
C09744=1191.760,23.696,-45.487,-179.616,5.756,148.906
C09745=1191.764,23.446,-45.472,-179.619,5.755,148.906
C09746=1191.770,23.196,-45.457,-179.621,5.754,148.907
C09747=1191.775,22.947,-45.442,-179.623,5.754,148.908
C09748=1191.780,22.698,-45.428,-179.626,5.753,148.908
C09749=1191.785,22.448,-45.412,-179.629,5.753,148.909
C09750=1191.790,22.199,-45.398,-179.631,5.752,148.909
C09751=1191.795,21.949,-45.383,-179.633,5.752,148.910
C09752=1191.800,21.699,-45.368,-179.636,5.751,148.911
C09753=1191.805,21.450,-45.354,-179.639,5.751,148.911
C09754=1191.810,21.201,-45.339,-179.641,5.750,148.912
C09755=1191.815,20.951,-45.325,-179.644,5.749,148.913
C09756=1191.820,20.701,-45.309,-179.646,5.749,148.913
C09757=1191.825,20.452,-45.295,-179.649,5.748,148.914
C09758=1191.830,20.202,-45.280,-179.651,5.747,148.914
C09759=1191.835,19.953,-45.265,-179.654,5.747,148.915
C09760=1191.840,19.703,-45.251,-179.656,5.746,148.916
C09761=1191.845,19.454,-45.236,-179.659,5.746,148.916
C09762=1191.850,19.204,-45.221,-179.661,5.745,148.917
C09763=1191.856,18.955,-45.207,-179.664,5.744,148.918
C09764=1191.860,18.706,-45.192,-179.666,5.744,148.918
C09765=1191.866,18.456,-45.177,-179.669,5.743,148.919
C09766=1191.871,18.206,-45.163,-179.671,5.743,148.919
C09767=1191.876,17.957,-45.148,-179.674,5.742,148.920
C09768=1191.880,17.708,-45.134,-179.677,5.742,148.921
C09769=1191.885,17.458,-45.120,-179.679,5.741,148.921
C09770=1191.891,17.208,-45.104,-179.681,5.740,148.922
C09771=1191.896,16.959,-45.090,-179.684,5.740,148.923
C09772=1191.901,16.709,-45.076,-179.687,5.739,148.923
C09773=1191.906,16.459,-45.061,-179.689,5.738,148.924
C09774=1191.910,16.210,-45.046,-179.691,5.738,148.924
C09775=1191.915,15.960,-45.032,-179.694,5.737,148.925
C09776=1191.922,15.711,-45.017,-179.697,5.737,148.926
C09777=1191.927,15.461,-45.003,-179.699,5.736,148.926
C09778=1191.931,15.212,-44.988,-179.702,5.736,148.927
C09779=1191.936,14.963,-44.974,-179.704,5.735,148.928
C09780=1191.941,14.713,-44.960,-179.707,5.735,148.928
C09781=1191.946,14.463,-44.945,-179.709,5.734,148.929
C09782=1191.951,14.214,-44.930,-179.712,5.733,148.929
C09783=1191.956,13.964,-44.916,-179.714,5.733,148.930
C09784=1191.961,13.715,-44.902,-179.717,5.732,148.931
C09785=1191.967,13.465,-44.887,-179.719,5.731,148.931
C09786=1191.972,13.216,-44.873,-179.722,5.731,148.932
C09787=1191.977,12.966,-44.859,-179.724,5.730,148.933
C09788=1191.981,12.717,-44.844,-179.727,5.730,148.933
C09789=1191.986,12.467,-44.829,-179.729,5.729,148.934
C09790=1191.991,12.217,-44.815,-179.732,5.728,148.934
C09791=1191.997,11.968,-44.801,-179.735,5.728,148.935
C09792=1192.002,11.719,-44.787,-179.737,5.727,148.936
C09793=1192.007,11.469,-44.773,-179.739,5.727,148.936
C09794=1192.012,11.219,-44.758,-179.742,5.726,148.937
C09795=1192.017,10.970,-44.744,-179.745,5.726,148.938
C09796=1192.022,10.720,-44.730,-179.747,5.725,148.938
C09797=1192.027,10.471,-44.716,-179.750,5.725,148.939
C09798=1192.032,10.222,-44.701,-179.752,5.724,148.939
C09799=1192.037,9.972,-44.687,-179.755,5.723,148.940
C09800=1192.042,9.722,-44.672,-179.757,5.723,148.941
C09801=1192.047,9.473,-44.658,-179.760,5.722,148.942
C09802=1192.052,9.224,-44.644,-179.762,5.721,148.942
C09803=1192.057,8.974,-44.630,-179.765,5.721,148.943
C09804=1192.062,8.724,-44.616,-179.768,5.720,148.943
C09805=1192.067,8.475,-44.601,-179.770,5.720,148.944
C09806=1192.073,8.226,-44.588,-179.772,5.719,148.944
C09807=1192.078,7.976,-44.573,-179.775,5.719,148.945
C09808=1192.083,7.726,-44.559,-179.778,5.718,148.946
C09809=1192.088,7.476,-44.545,-179.780,5.718,148.947
C09810=1192.093,7.227,-44.530,-179.782,5.717,148.947
C09811=1192.098,6.978,-44.516,-179.785,5.716,148.948
C09812=1192.103,6.728,-44.502,-179.788,5.716,148.948
C09813=1192.108,6.478,-44.488,-179.790,5.716,148.949
C09814=1192.113,6.228,-44.474,-179.792,5.715,148.950
C09815=1192.119,5.979,-44.460,-179.795,5.715,148.950
C09816=1192.123,5.730,-44.447,-179.797,5.714,148.951
C09817=1192.128,5.480,-44.433,-179.800,5.714,148.952
C09818=1192.133,5.230,-44.418,-179.803,5.713,148.952
C09819=1192.139,4.981,-44.404,-179.805,5.712,148.953
C09820=1192.143,4.731,-44.390,-179.807,5.712,148.953
C09821=1192.148,4.482,-44.376,-179.810,5.712,148.954
C09822=1192.154,4.233,-44.362,-179.813,5.711,148.955
C09823=1192.159,3.983,-44.348,-179.815,5.710,148.955
C09824=1192.163,3.733,-44.335,-179.818,5.710,148.956
C09825=1192.168,3.483,-44.320,-179.820,5.709,148.957
C09826=1192.174,3.234,-44.306,-179.823,5.709,148.957
C09827=1192.179,2.965,-44.291,-179.826,5.708,148.958
C09828=1192.185,2.695,-44.276,-179.828,5.708,148.959
C09829=1192.190,2.427,-44.261,-179.831,5.707,148.959
C09830=1192.195,2.157,-44.246,-179.833,5.707,148.960
C09831=1192.201,1.908,-44.232,-179.836,5.706,148.961
C09832=1192.206,1.658,-44.218,-179.838,5.705,148.961
C09833=1192.210,1.408,-44.205,-179.841,5.705,148.962
C09834=1192.216,1.159,-44.191,-179.844,5.704,148.963
C09835=1192.221,0.910,-44.176,-179.846,5.704,148.963
C09836=1192.226,0.659,-44.163,-179.848,5.703,148.964
C09837=1192.232,0.410,-44.149,-179.851,5.703,148.964
C09838=1192.236,0.161,-44.135,-179.853,5.703,148.965
C09839=1192.241,-0.089,-44.121,-179.856,5.702,148.966
C09840=1192.247,-0.338,-44.108,-179.858,5.702,148.966
C09841=1192.252,-0.588,-44.093,-179.861,5.701,148.967
C09842=1192.257,-0.837,-44.080,-179.863,5.701,148.968
C09843=1192.262,-1.087,-44.067,-179.866,5.700,148.968
C09844=1192.267,-1.337,-44.052,-179.868,5.699,148.969
C09845=1192.272,-1.586,-44.038,-179.871,5.699,148.969
C09846=1192.278,-1.836,-44.025,-179.873,5.698,148.970
C09847=1192.282,-2.086,-44.011,-179.876,5.698,148.971
C09848=1192.287,-2.335,-43.997,-179.878,5.697,148.971
C09849=1192.293,-2.585,-43.984,-179.880,5.697,148.972
C09850=1192.297,-2.834,-43.970,-179.883,5.697,148.973
C09851=1192.302,-3.083,-43.956,-179.886,5.696,148.973
C09852=1192.308,-3.334,-43.943,-179.888,5.696,148.974
C09853=1192.312,-3.582,-43.929,-179.890,5.695,148.975
C09854=1192.317,-3.832,-43.915,-179.893,5.695,148.975
C09855=1192.323,-4.082,-43.902,-179.896,5.694,148.976
C09856=1192.328,-4.331,-43.887,-179.898,5.694,148.977
C09857=1192.333,-4.581,-43.875,-179.901,5.693,148.977
C09858=1192.338,-4.830,-43.861,-179.903,5.692,148.978
C09859=1192.344,-5.081,-43.847,-179.905,5.693,148.978
C09860=1192.348,-5.329,-43.834,-179.908,5.692,148.979
C09861=1192.353,-5.579,-43.819,-179.911,5.692,148.980
C09862=1192.358,-5.828,-43.807,-179.913,5.691,148.980
C09863=1192.363,-6.078,-43.793,-179.915,5.690,148.981
C09864=1192.369,-6.329,-43.779,-179.918,5.690,148.982
C09865=1192.374,-6.577,-43.766,-179.921,5.689,148.982
C09866=1192.379,-6.828,-43.752,-179.923,5.689,148.983
C09867=1192.384,-7.077,-43.738,-179.926,5.688,148.983
C09868=1192.389,-7.327,-43.725,-179.928,5.688,148.984
C09869=1192.394,-7.576,-43.711,-179.930,5.688,148.985
C09870=1192.399,-7.826,-43.698,-179.933,5.687,148.986
C09871=1192.404,-8.075,-43.684,-179.935,5.687,148.986
C09872=1192.410,-8.325,-43.671,-179.938,5.686,148.987
C09873=1192.415,-8.574,-43.658,-179.940,5.686,148.987
C09874=1192.420,-8.824,-43.644,-179.943,5.685,148.988
C09875=1192.424,-9.074,-43.631,-179.946,5.685,148.989
C09876=1192.430,-9.323,-43.617,-179.948,5.684,148.989
C09877=1192.434,-9.573,-43.604,-179.950,5.684,148.990
C09878=1192.440,-9.822,-43.590,-179.953,5.684,148.991
C09879=1192.445,-10.072,-43.577,-179.955,5.683,148.991
C09880=1192.450,-10.321,-43.563,-179.957,5.682,148.992
C09881=1192.455,-10.571,-43.550,-179.960,5.682,148.992
C09882=1192.460,-10.821,-43.537,-179.963,5.681,148.993
C09883=1192.465,-11.070,-43.523,-179.965,5.681,148.994
C09884=1192.471,-11.320,-43.510,-179.968,5.681,148.995
C09885=1192.476,-11.570,-43.497,-179.970,5.680,148.995
C09886=1192.481,-11.819,-43.483,-179.972,5.680,148.996
C09887=1192.486,-12.068,-43.470,-179.975,5.679,148.996
C09888=1192.491,-12.318,-43.457,-179.978,5.679,148.997
C09889=1192.497,-12.567,-43.443,-179.980,5.678,148.998
C09890=1192.501,-12.817,-43.430,-179.982,5.678,148.998
C09891=1192.507,-13.067,-43.417,-179.985,5.678,148.999
C09892=1192.511,-13.316,-43.404,-179.987,5.678,149.000
C09893=1192.517,-13.566,-43.390,-179.990,5.677,149.000
C09894=1192.522,-13.816,-43.377,-179.992,5.676,149.001
C09895=1192.526,-14.065,-43.364,-179.995,5.676,149.002
C09896=1192.532,-14.315,-43.351,-179.997,5.675,149.002
C09897=1192.537,-14.564,-43.338,180.000,5.675,149.003
C09898=1192.543,-14.814,-43.325,179.998,5.675,149.004
C09899=1192.547,-15.063,-43.311,179.996,5.674,149.004
C09900=1192.553,-15.313,-43.298,179.993,5.674,149.005
C09901=1192.557,-15.563,-43.285,179.990,5.673,149.005
C09902=1192.562,-15.812,-43.272,179.988,5.673,149.006
C09903=1192.567,-16.062,-43.258,179.986,5.672,149.007
C09904=1192.572,-16.311,-43.245,179.983,5.672,149.007
C09905=1192.578,-16.561,-43.232,179.981,5.672,149.008
C09906=1192.583,-16.811,-43.219,179.978,5.671,149.009
C09907=1192.588,-17.060,-43.207,179.976,5.671,149.009
C09908=1192.593,-17.310,-43.192,179.973,5.670,149.010
C09909=1192.598,-17.559,-43.180,179.971,5.670,149.011
C09910=1192.604,-17.809,-43.167,179.968,5.669,149.011
C09911=1192.608,-18.059,-43.154,179.966,5.669,149.012
C09912=1192.614,-18.308,-43.141,179.963,5.669,149.013
C09913=1192.619,-18.558,-43.128,179.961,5.668,149.013
C09914=1192.624,-18.808,-43.115,179.958,5.668,149.014
C09915=1192.629,-19.057,-43.102,179.956,5.667,149.014
C09916=1192.634,-19.307,-43.088,179.953,5.667,149.015
C09917=1192.639,-19.556,-43.075,179.952,5.667,149.016
C09918=1192.644,-19.806,-43.063,179.949,5.666,149.016
C09919=1192.649,-20.056,-43.049,179.946,5.666,149.017
C09920=1192.655,-20.305,-43.037,179.944,5.665,149.018
C09921=1192.660,-20.555,-43.024,179.941,5.665,149.018
C09922=1192.665,-20.805,-43.010,179.939,5.664,149.019
C09923=1192.670,-21.054,-42.998,179.937,5.664,149.020
C09924=1192.675,-21.304,-42.985,179.934,5.664,149.020
C09925=1192.680,-21.554,-42.972,179.931,5.663,149.021
C09926=1192.686,-21.803,-42.959,179.929,5.663,149.022
C09927=1192.691,-22.053,-42.946,179.927,5.662,149.022
C09928=1192.696,-22.303,-42.933,179.924,5.662,149.023
C09929=1192.701,-22.552,-42.920,179.922,5.662,149.024
C09930=1192.706,-22.802,-42.908,179.919,5.662,149.024
C09931=1192.712,-23.072,-42.893,179.916,5.661,149.025
C09932=1192.717,-23.341,-42.879,179.914,5.661,149.026
C09933=1192.723,-23.610,-42.865,179.911,5.660,149.026
C09934=1192.728,-23.880,-42.851,179.909,5.660,149.027
C09935=1192.733,-24.129,-42.839,179.906,5.659,149.027
C09936=1192.738,-24.379,-42.826,179.904,5.658,149.028
C09937=1192.744,-24.629,-42.813,179.902,5.659,149.029
C09938=1192.749,-24.879,-42.801,179.899,5.658,149.030
C09939=1192.754,-25.128,-42.788,179.896,5.658,149.030
C09940=1192.759,-25.378,-42.775,179.894,5.657,149.031
C09941=1192.764,-25.627,-42.763,179.891,5.657,149.031
C09942=1192.770,-25.877,-42.749,179.889,5.657,149.032
C09943=1192.774,-26.127,-42.736,179.887,5.656,149.033
C09944=1192.779,-26.376,-42.724,179.884,5.656,149.034
C09945=1192.784,-26.626,-42.711,179.882,5.655,149.034
C09946=1192.789,-26.875,-42.699,179.879,5.655,149.035
C09947=1192.795,-27.125,-42.685,179.877,5.655,149.035
C09948=1192.800,-27.375,-42.673,179.874,5.655,149.036
C09949=1192.805,-27.625,-42.661,179.872,5.654,149.037
C09950=1192.810,-27.874,-42.648,179.870,5.653,149.037
C09951=1192.815,-28.124,-42.635,179.867,5.653,149.038
C09952=1192.820,-28.373,-42.622,179.865,5.653,149.039
C09953=1192.825,-28.623,-42.610,179.862,5.653,149.039
C09954=1192.831,-28.873,-42.597,179.860,5.652,149.040
C09955=1192.836,-29.122,-42.585,179.857,5.651,149.040
C09956=1192.841,-29.372,-42.572,179.855,5.652,149.041
C09957=1192.846,-29.621,-42.559,179.853,5.651,149.042
C09958=1192.851,-29.871,-42.547,179.850,5.651,149.043
C09959=1192.857,-30.121,-42.535,179.848,5.650,149.043
C09960=1192.862,-30.370,-42.522,179.845,5.649,149.044
C09961=1192.866,-30.620,-42.509,179.843,5.650,149.044
C09962=1192.871,-30.869,-42.497,179.840,5.649,149.045
C09963=1192.877,-31.119,-42.484,179.838,5.649,149.046
C09964=1192.883,-31.369,-42.471,179.836,5.648,149.046
C09965=1192.888,-31.618,-42.459,179.834,5.648,149.047
C09966=1192.892,-31.868,-42.446,179.831,5.648,149.048
C09967=1192.898,-32.118,-42.434,179.828,5.647,149.048
C09968=1192.903,-32.367,-42.421,179.826,5.647,149.049
C09969=1192.908,-32.617,-42.409,179.823,5.646,149.050
C09970=1192.913,-32.866,-42.396,179.821,5.647,149.050
C09971=1192.919,-33.116,-42.384,179.819,5.646,149.051
C09972=1192.923,-33.366,-42.371,179.816,5.646,149.052
C09973=1192.928,-33.615,-42.359,179.814,5.645,149.052
C09974=1192.934,-33.865,-42.347,179.812,5.645,149.053
C09975=1192.939,-34.115,-42.334,179.809,5.645,149.054
C09976=1192.944,-34.364,-42.322,179.806,5.644,149.054
C09977=1192.949,-34.614,-42.310,179.804,5.644,149.055
C09978=1192.954,-34.864,-42.297,179.802,5.644,149.055
C09979=1192.959,-35.114,-42.285,179.799,5.643,149.056
C09980=1192.964,-35.363,-42.272,179.797,5.643,149.057
C09981=1192.970,-35.612,-42.260,179.794,5.642,149.058
C09982=1192.975,-35.862,-42.248,179.792,5.642,149.058
C09983=1192.980,-36.112,-42.235,179.790,5.642,149.059
C09984=1192.985,-36.361,-42.223,179.787,5.641,149.059
C09985=1192.991,-36.611,-42.211,179.785,5.641,149.060
C09986=1192.996,-36.860,-42.198,179.782,5.641,149.061
C09987=1193.001,-37.111,-42.186,179.780,5.641,149.061
C09988=1193.006,-37.360,-42.173,179.778,5.640,149.062
C09989=1193.011,-37.610,-42.161,179.775,5.640,149.063
C09990=1193.016,-37.860,-42.149,179.772,5.639,149.063
C09991=1193.022,-38.109,-42.137,179.771,5.639,149.064
C09992=1193.027,-38.359,-42.124,179.768,5.639,149.065
C09993=1193.032,-38.608,-42.113,179.765,5.638,149.065
C09994=1193.037,-38.858,-42.100,179.763,5.638,149.066
C09995=1193.042,-39.107,-42.088,179.761,5.638,149.067
C09996=1193.047,-39.357,-42.076,179.758,5.637,149.067
//INST
///DATE 2021/06/25 14:28
///ATTR SC,RW,RJ
////FRAME ROBOT
///GROUP1 RB1
NOP
MOVL C00000 V=800.0 PL=0
MOVL C00001 V=800.0 PL=0
MOVL C00002 V=800.0 PL=0
MOVL C00003 V=800.0 PL=0
MOVL C00004 V=800.0 PL=0
MOVL C00005 V=800.0 PL=0
MOVL C00006 V=800.0 PL=0
MOVL C00007 V=800.0 PL=0
MOVL C00008 V=800.0 PL=0
MOVL C00009 V=800.0 PL=0
MOVL C00010 V=800.0 PL=0
MOVL C00011 V=800.0 PL=0
MOVL C00012 V=800.0 PL=0
MOVL C00013 V=800.0 PL=0
MOVL C00014 V=800.0 PL=0
MOVL C00015 V=800.0 PL=0
MOVL C00016 V=800.0 PL=0
MOVL C00017 V=800.0 PL=0
MOVL C00018 V=800.0 PL=0
MOVL C00019 V=800.0 PL=0
MOVL C00020 V=800.0 PL=0
MOVL C00021 V=800.0 PL=0
MOVL C00022 V=800.0 PL=0
MOVL C00023 V=800.0 PL=0
MOVL C00024 V=800.0 PL=0
MOVL C00025 V=800.0 PL=0
MOVL C00026 V=800.0 PL=0
MOVL C00027 V=800.0 PL=0
MOVL C00028 V=800.0 PL=0
MOVL C00029 V=800.0 PL=0
MOVL C00030 V=800.0 PL=0
MOVL C00031 V=800.0 PL=0
MOVL C00032 V=800.0 PL=0
MOVL C00033 V=800.0 PL=0
MOVL C00034 V=800.0 PL=0
MOVL C00035 V=800.0 PL=0
MOVL C00036 V=800.0 PL=0
MOVL C00037 V=800.0 PL=0
MOVL C00038 V=800.0 PL=0
MOVL C00039 V=800.0 PL=0
MOVL C00040 V=800.0 PL=0
MOVL C00041 V=800.0 PL=0
MOVL C00042 V=800.0 PL=0
MOVL C00043 V=800.0 PL=0
MOVL C00044 V=800.0 PL=0
MOVL C00045 V=800.0 PL=0
MOVL C00046 V=800.0 PL=0
MOVL C00047 V=800.0 PL=0
MOVL C00048 V=800.0 PL=0
MOVL C00049 V=800.0 PL=0
MOVL C00050 V=800.0 PL=0
MOVL C00051 V=800.0 PL=0
MOVL C00052 V=800.0 PL=0
MOVL C00053 V=800.0 PL=0
MOVL C00054 V=800.0 PL=0
MOVL C00055 V=800.0 PL=0
MOVL C00056 V=800.0 PL=0
MOVL C00057 V=800.0 PL=0
MOVL C00058 V=800.0 PL=0
MOVL C00059 V=800.0 PL=0
MOVL C00060 V=800.0 PL=0
MOVL C00061 V=800.0 PL=0
MOVL C00062 V=800.0 PL=0
MOVL C00063 V=800.0 PL=0
MOVL C00064 V=800.0 PL=0
MOVL C00065 V=800.0 PL=0
MOVL C00066 V=800.0 PL=0
MOVL C00067 V=800.0 PL=0
MOVL C00068 V=800.0 PL=0
MOVL C00069 V=800.0 PL=0
MOVL C00070 V=800.0 PL=0
MOVL C00071 V=800.0 PL=0
MOVL C00072 V=800.0 PL=0
MOVL C00073 V=800.0 PL=0
MOVL C00074 V=800.0 PL=0
MOVL C00075 V=800.0 PL=0
MOVL C00076 V=800.0 PL=0
MOVL C00077 V=800.0 PL=0
MOVL C00078 V=800.0 PL=0
MOVL C00079 V=800.0 PL=0
MOVL C00080 V=800.0 PL=0
MOVL C00081 V=800.0 PL=0
MOVL C00082 V=800.0 PL=0
MOVL C00083 V=800.0 PL=0
MOVL C00084 V=800.0 PL=0
MOVL C00085 V=800.0 PL=0
MOVL C00086 V=800.0 PL=0
MOVL C00087 V=800.0 PL=0
MOVL C00088 V=800.0 PL=0
MOVL C00089 V=800.0 PL=0
MOVL C00090 V=800.0 PL=0
MOVL C00091 V=800.0 PL=0
MOVL C00092 V=800.0 PL=0
MOVL C00093 V=800.0 PL=0
MOVL C00094 V=800.0 PL=0
MOVL C00095 V=800.0 PL=0
MOVL C00096 V=800.0 PL=0
MOVL C00097 V=800.0 PL=0
MOVL C00098 V=800.0 PL=0
MOVL C00099 V=800.0 PL=0
MOVL C00100 V=800.0 PL=0
MOVL C00101 V=800.0 PL=0
MOVL C00102 V=800.0 PL=0
MOVL C00103 V=800.0 PL=0
MOVL C00104 V=800.0 PL=0
MOVL C00105 V=800.0 PL=0
MOVL C00106 V=800.0 PL=0
MOVL C00107 V=800.0 PL=0
MOVL C00108 V=800.0 PL=0
MOVL C00109 V=800.0 PL=0
MOVL C00110 V=800.0 PL=0
MOVL C00111 V=800.0 PL=0
MOVL C00112 V=800.0 PL=0
MOVL C00113 V=800.0 PL=0
MOVL C00114 V=800.0 PL=0
MOVL C00115 V=800.0 PL=0
MOVL C00116 V=800.0 PL=0
MOVL C00117 V=800.0 PL=0
MOVL C00118 V=800.0 PL=0
MOVL C00119 V=800.0 PL=0
MOVL C00120 V=800.0 PL=0
MOVL C00121 V=800.0 PL=0
MOVL C00122 V=800.0 PL=0
MOVL C00123 V=800.0 PL=0
MOVL C00124 V=800.0 PL=0
MOVL C00125 V=800.0 PL=0
MOVL C00126 V=800.0 PL=0
MOVL C00127 V=800.0 PL=0
MOVL C00128 V=800.0 PL=0
MOVL C00129 V=800.0 PL=0
MOVL C00130 V=800.0 PL=0
MOVL C00131 V=800.0 PL=0
MOVL C00132 V=800.0 PL=0
MOVL C00133 V=800.0 PL=0
MOVL C00134 V=800.0 PL=0
MOVL C00135 V=800.0 PL=0
MOVL C00136 V=800.0 PL=0
MOVL C00137 V=800.0 PL=0
MOVL C00138 V=800.0 PL=0
MOVL C00139 V=800.0 PL=0
MOVL C00140 V=800.0 PL=0
MOVL C00141 V=800.0 PL=0
MOVL C00142 V=800.0 PL=0
MOVL C00143 V=800.0 PL=0
MOVL C00144 V=800.0 PL=0
MOVL C00145 V=800.0 PL=0
MOVL C00146 V=800.0 PL=0
MOVL C00147 V=800.0 PL=0
MOVL C00148 V=800.0 PL=0
MOVL C00149 V=800.0 PL=0
MOVL C00150 V=800.0 PL=0
MOVL C00151 V=800.0 PL=0
MOVL C00152 V=800.0 PL=0
MOVL C00153 V=800.0 PL=0
MOVL C00154 V=800.0 PL=0
MOVL C00155 V=800.0 PL=0
MOVL C00156 V=800.0 PL=0
MOVL C00157 V=800.0 PL=0
MOVL C00158 V=800.0 PL=0
MOVL C00159 V=800.0 PL=0
MOVL C00160 V=800.0 PL=0
MOVL C00161 V=800.0 PL=0
MOVL C00162 V=800.0 PL=0
MOVL C00163 V=800.0 PL=0
MOVL C00164 V=800.0 PL=0
MOVL C00165 V=800.0 PL=0
MOVL C00166 V=800.0 PL=0
MOVL C00167 V=800.0 PL=0
MOVL C00168 V=800.0 PL=0
MOVL C00169 V=800.0 PL=0
MOVL C00170 V=800.0 PL=0
MOVL C00171 V=800.0 PL=0
MOVL C00172 V=800.0 PL=0
MOVL C00173 V=800.0 PL=0
MOVL C00174 V=800.0 PL=0
MOVL C00175 V=800.0 PL=0
MOVL C00176 V=800.0 PL=0
MOVL C00177 V=800.0 PL=0
MOVL C00178 V=800.0 PL=0
MOVL C00179 V=800.0 PL=0
MOVL C00180 V=800.0 PL=0
MOVL C00181 V=800.0 PL=0
MOVL C00182 V=800.0 PL=0
MOVL C00183 V=800.0 PL=0
MOVL C00184 V=800.0 PL=0
MOVL C00185 V=800.0 PL=0
MOVL C00186 V=800.0 PL=0
MOVL C00187 V=800.0 PL=0
MOVL C00188 V=800.0 PL=0
MOVL C00189 V=800.0 PL=0
MOVL C00190 V=800.0 PL=0
MOVL C00191 V=800.0 PL=0
MOVL C00192 V=800.0 PL=0
MOVL C00193 V=800.0 PL=0
MOVL C00194 V=800.0 PL=0
MOVL C00195 V=800.0 PL=0
MOVL C00196 V=800.0 PL=0
MOVL C00197 V=800.0 PL=0
MOVL C00198 V=800.0 PL=0
MOVL C00199 V=800.0 PL=0
MOVL C00200 V=800.0 PL=0
MOVL C00201 V=800.0 PL=0
MOVL C00202 V=800.0 PL=0
MOVL C00203 V=800.0 PL=0
MOVL C00204 V=800.0 PL=0
MOVL C00205 V=800.0 PL=0
MOVL C00206 V=800.0 PL=0
MOVL C00207 V=800.0 PL=0
MOVL C00208 V=800.0 PL=0
MOVL C00209 V=800.0 PL=0
MOVL C00210 V=800.0 PL=0
MOVL C00211 V=800.0 PL=0
MOVL C00212 V=800.0 PL=0
MOVL C00213 V=800.0 PL=0
MOVL C00214 V=800.0 PL=0
MOVL C00215 V=800.0 PL=0
MOVL C00216 V=800.0 PL=0
MOVL C00217 V=800.0 PL=0
MOVL C00218 V=800.0 PL=0
MOVL C00219 V=800.0 PL=0
MOVL C00220 V=800.0 PL=0
MOVL C00221 V=800.0 PL=0
MOVL C00222 V=800.0 PL=0
MOVL C00223 V=800.0 PL=0
MOVL C00224 V=800.0 PL=0
MOVL C00225 V=800.0 PL=0
MOVL C00226 V=800.0 PL=0
MOVL C00227 V=800.0 PL=0
MOVL C00228 V=800.0 PL=0
MOVL C00229 V=800.0 PL=0
MOVL C00230 V=800.0 PL=0
MOVL C00231 V=800.0 PL=0
MOVL C00232 V=800.0 PL=0
MOVL C00233 V=800.0 PL=0
MOVL C00234 V=800.0 PL=0
MOVL C00235 V=800.0 PL=0
MOVL C00236 V=800.0 PL=0
MOVL C00237 V=800.0 PL=0
MOVL C00238 V=800.0 PL=0
MOVL C00239 V=800.0 PL=0
MOVL C00240 V=800.0 PL=0
MOVL C00241 V=800.0 PL=0
MOVL C00242 V=800.0 PL=0
MOVL C00243 V=800.0 PL=0
MOVL C00244 V=800.0 PL=0
MOVL C00245 V=800.0 PL=0
MOVL C00246 V=800.0 PL=0
MOVL C00247 V=800.0 PL=0
MOVL C00248 V=800.0 PL=0
MOVL C00249 V=800.0 PL=0
MOVL C00250 V=800.0 PL=0
MOVL C00251 V=800.0 PL=0
MOVL C00252 V=800.0 PL=0
MOVL C00253 V=800.0 PL=0
MOVL C00254 V=800.0 PL=0
MOVL C00255 V=800.0 PL=0
MOVL C00256 V=800.0 PL=0
MOVL C00257 V=800.0 PL=0
MOVL C00258 V=800.0 PL=0
MOVL C00259 V=800.0 PL=0
MOVL C00260 V=800.0 PL=0
MOVL C00261 V=800.0 PL=0
MOVL C00262 V=800.0 PL=0
MOVL C00263 V=800.0 PL=0
MOVL C00264 V=800.0 PL=0
MOVL C00265 V=800.0 PL=0
MOVL C00266 V=800.0 PL=0
MOVL C00267 V=800.0 PL=0
MOVL C00268 V=800.0 PL=0
MOVL C00269 V=800.0 PL=0
MOVL C00270 V=800.0 PL=0
MOVL C00271 V=800.0 PL=0
MOVL C00272 V=800.0 PL=0
MOVL C00273 V=800.0 PL=0
MOVL C00274 V=800.0 PL=0
MOVL C00275 V=800.0 PL=0
MOVL C00276 V=800.0 PL=0
MOVL C00277 V=800.0 PL=0
MOVL C00278 V=800.0 PL=0
MOVL C00279 V=800.0 PL=0
MOVL C00280 V=800.0 PL=0
MOVL C00281 V=800.0 PL=0
MOVL C00282 V=800.0 PL=0
MOVL C00283 V=800.0 PL=0
MOVL C00284 V=800.0 PL=0
MOVL C00285 V=800.0 PL=0
MOVL C00286 V=800.0 PL=0
MOVL C00287 V=800.0 PL=0
MOVL C00288 V=800.0 PL=0
MOVL C00289 V=800.0 PL=0
MOVL C00290 V=800.0 PL=0
MOVL C00291 V=800.0 PL=0
MOVL C00292 V=800.0 PL=0
MOVL C00293 V=800.0 PL=0
MOVL C00294 V=800.0 PL=0
MOVL C00295 V=800.0 PL=0
MOVL C00296 V=800.0 PL=0
MOVL C00297 V=800.0 PL=0
MOVL C00298 V=800.0 PL=0
MOVL C00299 V=800.0 PL=0
MOVL C00300 V=800.0 PL=0
MOVL C00301 V=800.0 PL=0
MOVL C00302 V=800.0 PL=0
MOVL C00303 V=800.0 PL=0
MOVL C00304 V=800.0 PL=0
MOVL C00305 V=800.0 PL=0
MOVL C00306 V=800.0 PL=0
MOVL C00307 V=800.0 PL=0
MOVL C00308 V=800.0 PL=0
MOVL C00309 V=800.0 PL=0
MOVL C00310 V=800.0 PL=0
MOVL C00311 V=800.0 PL=0
MOVL C00312 V=800.0 PL=0
MOVL C00313 V=800.0 PL=0
MOVL C00314 V=800.0 PL=0
MOVL C00315 V=800.0 PL=0
MOVL C00316 V=800.0 PL=0
MOVL C00317 V=800.0 PL=0
MOVL C00318 V=800.0 PL=0
MOVL C00319 V=800.0 PL=0
MOVL C00320 V=800.0 PL=0
MOVL C00321 V=800.0 PL=0
MOVL C00322 V=800.0 PL=0
MOVL C00323 V=800.0 PL=0
MOVL C00324 V=800.0 PL=0
MOVL C00325 V=800.0 PL=0
MOVL C00326 V=800.0 PL=0
MOVL C00327 V=800.0 PL=0
MOVL C00328 V=800.0 PL=0
MOVL C00329 V=800.0 PL=0
MOVL C00330 V=800.0 PL=0
MOVL C00331 V=800.0 PL=0
MOVL C00332 V=800.0 PL=0
MOVL C00333 V=800.0 PL=0
MOVL C00334 V=800.0 PL=0
MOVL C00335 V=800.0 PL=0
MOVL C00336 V=800.0 PL=0
MOVL C00337 V=800.0 PL=0
MOVL C00338 V=800.0 PL=0
MOVL C00339 V=800.0 PL=0
MOVL C00340 V=800.0 PL=0
MOVL C00341 V=800.0 PL=0
MOVL C00342 V=800.0 PL=0
MOVL C00343 V=800.0 PL=0
MOVL C00344 V=800.0 PL=0
MOVL C00345 V=800.0 PL=0
MOVL C00346 V=800.0 PL=0
MOVL C00347 V=800.0 PL=0
MOVL C00348 V=800.0 PL=0
MOVL C00349 V=800.0 PL=0
MOVL C00350 V=800.0 PL=0
MOVL C00351 V=800.0 PL=0
MOVL C00352 V=800.0 PL=0
MOVL C00353 V=800.0 PL=0
MOVL C00354 V=800.0 PL=0
MOVL C00355 V=800.0 PL=0
MOVL C00356 V=800.0 PL=0
MOVL C00357 V=800.0 PL=0
MOVL C00358 V=800.0 PL=0
MOVL C00359 V=800.0 PL=0
MOVL C00360 V=800.0 PL=0
MOVL C00361 V=800.0 PL=0
MOVL C00362 V=800.0 PL=0
MOVL C00363 V=800.0 PL=0
MOVL C00364 V=800.0 PL=0
MOVL C00365 V=800.0 PL=0
MOVL C00366 V=800.0 PL=0
MOVL C00367 V=800.0 PL=0
MOVL C00368 V=800.0 PL=0
MOVL C00369 V=800.0 PL=0
MOVL C00370 V=800.0 PL=0
MOVL C00371 V=800.0 PL=0
MOVL C00372 V=800.0 PL=0
MOVL C00373 V=800.0 PL=0
MOVL C00374 V=800.0 PL=0
MOVL C00375 V=800.0 PL=0
MOVL C00376 V=800.0 PL=0
MOVL C00377 V=800.0 PL=0
MOVL C00378 V=800.0 PL=0
MOVL C00379 V=800.0 PL=0
MOVL C00380 V=800.0 PL=0
MOVL C00381 V=800.0 PL=0
MOVL C00382 V=800.0 PL=0
MOVL C00383 V=800.0 PL=0
MOVL C00384 V=800.0 PL=0
MOVL C00385 V=800.0 PL=0
MOVL C00386 V=800.0 PL=0
MOVL C00387 V=800.0 PL=0
MOVL C00388 V=800.0 PL=0
MOVL C00389 V=800.0 PL=0
MOVL C00390 V=800.0 PL=0
MOVL C00391 V=800.0 PL=0
MOVL C00392 V=800.0 PL=0
MOVL C00393 V=800.0 PL=0
MOVL C00394 V=800.0 PL=0
MOVL C00395 V=800.0 PL=0
MOVL C00396 V=800.0 PL=0
MOVL C00397 V=800.0 PL=0
MOVL C00398 V=800.0 PL=0
MOVL C00399 V=800.0 PL=0
MOVL C00400 V=800.0 PL=0
MOVL C00401 V=800.0 PL=0
MOVL C00402 V=800.0 PL=0
MOVL C00403 V=800.0 PL=0
MOVL C00404 V=800.0 PL=0
MOVL C00405 V=800.0 PL=0
MOVL C00406 V=800.0 PL=0
MOVL C00407 V=800.0 PL=0
MOVL C00408 V=800.0 PL=0
MOVL C00409 V=800.0 PL=0
MOVL C00410 V=800.0 PL=0
MOVL C00411 V=800.0 PL=0
MOVL C00412 V=800.0 PL=0
MOVL C00413 V=800.0 PL=0
MOVL C00414 V=800.0 PL=0
MOVL C00415 V=800.0 PL=0
MOVL C00416 V=800.0 PL=0
MOVL C00417 V=800.0 PL=0
MOVL C00418 V=800.0 PL=0
MOVL C00419 V=800.0 PL=0
MOVL C00420 V=800.0 PL=0
MOVL C00421 V=800.0 PL=0
MOVL C00422 V=800.0 PL=0
MOVL C00423 V=800.0 PL=0
MOVL C00424 V=800.0 PL=0
MOVL C00425 V=800.0 PL=0
MOVL C00426 V=800.0 PL=0
MOVL C00427 V=800.0 PL=0
MOVL C00428 V=800.0 PL=0
MOVL C00429 V=800.0 PL=0
MOVL C00430 V=800.0 PL=0
MOVL C00431 V=800.0 PL=0
MOVL C00432 V=800.0 PL=0
MOVL C00433 V=800.0 PL=0
MOVL C00434 V=800.0 PL=0
MOVL C00435 V=800.0 PL=0
MOVL C00436 V=800.0 PL=0
MOVL C00437 V=800.0 PL=0
MOVL C00438 V=800.0 PL=0
MOVL C00439 V=800.0 PL=0
MOVL C00440 V=800.0 PL=0
MOVL C00441 V=800.0 PL=0
MOVL C00442 V=800.0 PL=0
MOVL C00443 V=800.0 PL=0
MOVL C00444 V=800.0 PL=0
MOVL C00445 V=800.0 PL=0
MOVL C00446 V=800.0 PL=0
MOVL C00447 V=800.0 PL=0
MOVL C00448 V=800.0 PL=0
MOVL C00449 V=800.0 PL=0
MOVL C00450 V=800.0 PL=0
MOVL C00451 V=800.0 PL=0
MOVL C00452 V=800.0 PL=0
MOVL C00453 V=800.0 PL=0
MOVL C00454 V=800.0 PL=0
MOVL C00455 V=800.0 PL=0
MOVL C00456 V=800.0 PL=0
MOVL C00457 V=800.0 PL=0
MOVL C00458 V=800.0 PL=0
MOVL C00459 V=800.0 PL=0
MOVL C00460 V=800.0 PL=0
MOVL C00461 V=800.0 PL=0
MOVL C00462 V=800.0 PL=0
MOVL C00463 V=800.0 PL=0
MOVL C00464 V=800.0 PL=0
MOVL C00465 V=800.0 PL=0
MOVL C00466 V=800.0 PL=0
MOVL C00467 V=800.0 PL=0
MOVL C00468 V=800.0 PL=0
MOVL C00469 V=800.0 PL=0
MOVL C00470 V=800.0 PL=0
MOVL C00471 V=800.0 PL=0
MOVL C00472 V=800.0 PL=0
MOVL C00473 V=800.0 PL=0
MOVL C00474 V=800.0 PL=0
MOVL C00475 V=800.0 PL=0
MOVL C00476 V=800.0 PL=0
MOVL C00477 V=800.0 PL=0
MOVL C00478 V=800.0 PL=0
MOVL C00479 V=800.0 PL=0
MOVL C00480 V=800.0 PL=0
MOVL C00481 V=800.0 PL=0
MOVL C00482 V=800.0 PL=0
MOVL C00483 V=800.0 PL=0
MOVL C00484 V=800.0 PL=0
MOVL C00485 V=800.0 PL=0
MOVL C00486 V=800.0 PL=0
MOVL C00487 V=800.0 PL=0
MOVL C00488 V=800.0 PL=0
MOVL C00489 V=800.0 PL=0
MOVL C00490 V=800.0 PL=0
MOVL C00491 V=800.0 PL=0
MOVL C00492 V=800.0 PL=0
MOVL C00493 V=800.0 PL=0
MOVL C00494 V=800.0 PL=0
MOVL C00495 V=800.0 PL=0
MOVL C00496 V=800.0 PL=0
MOVL C00497 V=800.0 PL=0
MOVL C00498 V=800.0 PL=0
MOVL C00499 V=800.0 PL=0
MOVL C00500 V=800.0 PL=0
MOVL C00501 V=800.0 PL=0
MOVL C00502 V=800.0 PL=0
MOVL C00503 V=800.0 PL=0
MOVL C00504 V=800.0 PL=0
MOVL C00505 V=800.0 PL=0
MOVL C00506 V=800.0 PL=0
MOVL C00507 V=800.0 PL=0
MOVL C00508 V=800.0 PL=0
MOVL C00509 V=800.0 PL=0
MOVL C00510 V=800.0 PL=0
MOVL C00511 V=800.0 PL=0
MOVL C00512 V=800.0 PL=0
MOVL C00513 V=800.0 PL=0
MOVL C00514 V=800.0 PL=0
MOVL C00515 V=800.0 PL=0
MOVL C00516 V=800.0 PL=0
MOVL C00517 V=800.0 PL=0
MOVL C00518 V=800.0 PL=0
MOVL C00519 V=800.0 PL=0
MOVL C00520 V=800.0 PL=0
MOVL C00521 V=800.0 PL=0
MOVL C00522 V=800.0 PL=0
MOVL C00523 V=800.0 PL=0
MOVL C00524 V=800.0 PL=0
MOVL C00525 V=800.0 PL=0
MOVL C00526 V=800.0 PL=0
MOVL C00527 V=800.0 PL=0
MOVL C00528 V=800.0 PL=0
MOVL C00529 V=800.0 PL=0
MOVL C00530 V=800.0 PL=0
MOVL C00531 V=800.0 PL=0
MOVL C00532 V=800.0 PL=0
MOVL C00533 V=800.0 PL=0
MOVL C00534 V=800.0 PL=0
MOVL C00535 V=800.0 PL=0
MOVL C00536 V=800.0 PL=0
MOVL C00537 V=800.0 PL=0
MOVL C00538 V=800.0 PL=0
MOVL C00539 V=800.0 PL=0
MOVL C00540 V=800.0 PL=0
MOVL C00541 V=800.0 PL=0
MOVL C00542 V=800.0 PL=0
MOVL C00543 V=800.0 PL=0
MOVL C00544 V=800.0 PL=0
MOVL C00545 V=800.0 PL=0
MOVL C00546 V=800.0 PL=0
MOVL C00547 V=800.0 PL=0
MOVL C00548 V=800.0 PL=0
MOVL C00549 V=800.0 PL=0
MOVL C00550 V=800.0 PL=0
MOVL C00551 V=800.0 PL=0
MOVL C00552 V=800.0 PL=0
MOVL C00553 V=800.0 PL=0
MOVL C00554 V=800.0 PL=0
MOVL C00555 V=800.0 PL=0
MOVL C00556 V=800.0 PL=0
MOVL C00557 V=800.0 PL=0
MOVL C00558 V=800.0 PL=0
MOVL C00559 V=800.0 PL=0
MOVL C00560 V=800.0 PL=0
MOVL C00561 V=800.0 PL=0
MOVL C00562 V=800.0 PL=0
MOVL C00563 V=800.0 PL=0
MOVL C00564 V=800.0 PL=0
MOVL C00565 V=800.0 PL=0
MOVL C00566 V=800.0 PL=0
MOVL C00567 V=800.0 PL=0
MOVL C00568 V=800.0 PL=0
MOVL C00569 V=800.0 PL=0
MOVL C00570 V=800.0 PL=0
MOVL C00571 V=800.0 PL=0
MOVL C00572 V=800.0 PL=0
MOVL C00573 V=800.0 PL=0
MOVL C00574 V=800.0 PL=0
MOVL C00575 V=800.0 PL=0
MOVL C00576 V=800.0 PL=0
MOVL C00577 V=800.0 PL=0
MOVL C00578 V=800.0 PL=0
MOVL C00579 V=800.0 PL=0
MOVL C00580 V=800.0 PL=0
MOVL C00581 V=800.0 PL=0
MOVL C00582 V=800.0 PL=0
MOVL C00583 V=800.0 PL=0
MOVL C00584 V=800.0 PL=0
MOVL C00585 V=800.0 PL=0
MOVL C00586 V=800.0 PL=0
MOVL C00587 V=800.0 PL=0
MOVL C00588 V=800.0 PL=0
MOVL C00589 V=800.0 PL=0
MOVL C00590 V=800.0 PL=0
MOVL C00591 V=800.0 PL=0
MOVL C00592 V=800.0 PL=0
MOVL C00593 V=800.0 PL=0
MOVL C00594 V=800.0 PL=0
MOVL C00595 V=800.0 PL=0
MOVL C00596 V=800.0 PL=0
MOVL C00597 V=800.0 PL=0
MOVL C00598 V=800.0 PL=0
MOVL C00599 V=800.0 PL=0
MOVL C00600 V=800.0 PL=0
MOVL C00601 V=800.0 PL=0
MOVL C00602 V=800.0 PL=0
MOVL C00603 V=800.0 PL=0
MOVL C00604 V=800.0 PL=0
MOVL C00605 V=800.0 PL=0
MOVL C00606 V=800.0 PL=0
MOVL C00607 V=800.0 PL=0
MOVL C00608 V=800.0 PL=0
MOVL C00609 V=800.0 PL=0
MOVL C00610 V=800.0 PL=0
MOVL C00611 V=800.0 PL=0
MOVL C00612 V=800.0 PL=0
MOVL C00613 V=800.0 PL=0
MOVL C00614 V=800.0 PL=0
MOVL C00615 V=800.0 PL=0
MOVL C00616 V=800.0 PL=0
MOVL C00617 V=800.0 PL=0
MOVL C00618 V=800.0 PL=0
MOVL C00619 V=800.0 PL=0
MOVL C00620 V=800.0 PL=0
MOVL C00621 V=800.0 PL=0
MOVL C00622 V=800.0 PL=0
MOVL C00623 V=800.0 PL=0
MOVL C00624 V=800.0 PL=0
MOVL C00625 V=800.0 PL=0
MOVL C00626 V=800.0 PL=0
MOVL C00627 V=800.0 PL=0
MOVL C00628 V=800.0 PL=0
MOVL C00629 V=800.0 PL=0
MOVL C00630 V=800.0 PL=0
MOVL C00631 V=800.0 PL=0
MOVL C00632 V=800.0 PL=0
MOVL C00633 V=800.0 PL=0
MOVL C00634 V=800.0 PL=0
MOVL C00635 V=800.0 PL=0
MOVL C00636 V=800.0 PL=0
MOVL C00637 V=800.0 PL=0
MOVL C00638 V=800.0 PL=0
MOVL C00639 V=800.0 PL=0
MOVL C00640 V=800.0 PL=0
MOVL C00641 V=800.0 PL=0
MOVL C00642 V=800.0 PL=0
MOVL C00643 V=800.0 PL=0
MOVL C00644 V=800.0 PL=0
MOVL C00645 V=800.0 PL=0
MOVL C00646 V=800.0 PL=0
MOVL C00647 V=800.0 PL=0
MOVL C00648 V=800.0 PL=0
MOVL C00649 V=800.0 PL=0
MOVL C00650 V=800.0 PL=0
MOVL C00651 V=800.0 PL=0
MOVL C00652 V=800.0 PL=0
MOVL C00653 V=800.0 PL=0
MOVL C00654 V=800.0 PL=0
MOVL C00655 V=800.0 PL=0
MOVL C00656 V=800.0 PL=0
MOVL C00657 V=800.0 PL=0
MOVL C00658 V=800.0 PL=0
MOVL C00659 V=800.0 PL=0
MOVL C00660 V=800.0 PL=0
MOVL C00661 V=800.0 PL=0
MOVL C00662 V=800.0 PL=0
MOVL C00663 V=800.0 PL=0
MOVL C00664 V=800.0 PL=0
MOVL C00665 V=800.0 PL=0
MOVL C00666 V=800.0 PL=0
MOVL C00667 V=800.0 PL=0
MOVL C00668 V=800.0 PL=0
MOVL C00669 V=800.0 PL=0
MOVL C00670 V=800.0 PL=0
MOVL C00671 V=800.0 PL=0
MOVL C00672 V=800.0 PL=0
MOVL C00673 V=800.0 PL=0
MOVL C00674 V=800.0 PL=0
MOVL C00675 V=800.0 PL=0
MOVL C00676 V=800.0 PL=0
MOVL C00677 V=800.0 PL=0
MOVL C00678 V=800.0 PL=0
MOVL C00679 V=800.0 PL=0
MOVL C00680 V=800.0 PL=0
MOVL C00681 V=800.0 PL=0
MOVL C00682 V=800.0 PL=0
MOVL C00683 V=800.0 PL=0
MOVL C00684 V=800.0 PL=0
MOVL C00685 V=800.0 PL=0
MOVL C00686 V=800.0 PL=0
MOVL C00687 V=800.0 PL=0
MOVL C00688 V=800.0 PL=0
MOVL C00689 V=800.0 PL=0
MOVL C00690 V=800.0 PL=0
MOVL C00691 V=800.0 PL=0
MOVL C00692 V=800.0 PL=0
MOVL C00693 V=800.0 PL=0
MOVL C00694 V=800.0 PL=0
MOVL C00695 V=800.0 PL=0
MOVL C00696 V=800.0 PL=0
MOVL C00697 V=800.0 PL=0
MOVL C00698 V=800.0 PL=0
MOVL C00699 V=800.0 PL=0
MOVL C00700 V=800.0 PL=0
MOVL C00701 V=800.0 PL=0
MOVL C00702 V=800.0 PL=0
MOVL C00703 V=800.0 PL=0
MOVL C00704 V=800.0 PL=0
MOVL C00705 V=800.0 PL=0
MOVL C00706 V=800.0 PL=0
MOVL C00707 V=800.0 PL=0
MOVL C00708 V=800.0 PL=0
MOVL C00709 V=800.0 PL=0
MOVL C00710 V=800.0 PL=0
MOVL C00711 V=800.0 PL=0
MOVL C00712 V=800.0 PL=0
MOVL C00713 V=800.0 PL=0
MOVL C00714 V=800.0 PL=0
MOVL C00715 V=800.0 PL=0
MOVL C00716 V=800.0 PL=0
MOVL C00717 V=800.0 PL=0
MOVL C00718 V=800.0 PL=0
MOVL C00719 V=800.0 PL=0
MOVL C00720 V=800.0 PL=0
MOVL C00721 V=800.0 PL=0
MOVL C00722 V=800.0 PL=0
MOVL C00723 V=800.0 PL=0
MOVL C00724 V=800.0 PL=0
MOVL C00725 V=800.0 PL=0
MOVL C00726 V=800.0 PL=0
MOVL C00727 V=800.0 PL=0
MOVL C00728 V=800.0 PL=0
MOVL C00729 V=800.0 PL=0
MOVL C00730 V=800.0 PL=0
MOVL C00731 V=800.0 PL=0
MOVL C00732 V=800.0 PL=0
MOVL C00733 V=800.0 PL=0
MOVL C00734 V=800.0 PL=0
MOVL C00735 V=800.0 PL=0
MOVL C00736 V=800.0 PL=0
MOVL C00737 V=800.0 PL=0
MOVL C00738 V=800.0 PL=0
MOVL C00739 V=800.0 PL=0
MOVL C00740 V=800.0 PL=0
MOVL C00741 V=800.0 PL=0
MOVL C00742 V=800.0 PL=0
MOVL C00743 V=800.0 PL=0
MOVL C00744 V=800.0 PL=0
MOVL C00745 V=800.0 PL=0
MOVL C00746 V=800.0 PL=0
MOVL C00747 V=800.0 PL=0
MOVL C00748 V=800.0 PL=0
MOVL C00749 V=800.0 PL=0
MOVL C00750 V=800.0 PL=0
MOVL C00751 V=800.0 PL=0
MOVL C00752 V=800.0 PL=0
MOVL C00753 V=800.0 PL=0
MOVL C00754 V=800.0 PL=0
MOVL C00755 V=800.0 PL=0
MOVL C00756 V=800.0 PL=0
MOVL C00757 V=800.0 PL=0
MOVL C00758 V=800.0 PL=0
MOVL C00759 V=800.0 PL=0
MOVL C00760 V=800.0 PL=0
MOVL C00761 V=800.0 PL=0
MOVL C00762 V=800.0 PL=0
MOVL C00763 V=800.0 PL=0
MOVL C00764 V=800.0 PL=0
MOVL C00765 V=800.0 PL=0
MOVL C00766 V=800.0 PL=0
MOVL C00767 V=800.0 PL=0
MOVL C00768 V=800.0 PL=0
MOVL C00769 V=800.0 PL=0
MOVL C00770 V=800.0 PL=0
MOVL C00771 V=800.0 PL=0
MOVL C00772 V=800.0 PL=0
MOVL C00773 V=800.0 PL=0
MOVL C00774 V=800.0 PL=0
MOVL C00775 V=800.0 PL=0
MOVL C00776 V=800.0 PL=0
MOVL C00777 V=800.0 PL=0
MOVL C00778 V=800.0 PL=0
MOVL C00779 V=800.0 PL=0
MOVL C00780 V=800.0 PL=0
MOVL C00781 V=800.0 PL=0
MOVL C00782 V=800.0 PL=0
MOVL C00783 V=800.0 PL=0
MOVL C00784 V=800.0 PL=0
MOVL C00785 V=800.0 PL=0
MOVL C00786 V=800.0 PL=0
MOVL C00787 V=800.0 PL=0
MOVL C00788 V=800.0 PL=0
MOVL C00789 V=800.0 PL=0
MOVL C00790 V=800.0 PL=0
MOVL C00791 V=800.0 PL=0
MOVL C00792 V=800.0 PL=0
MOVL C00793 V=800.0 PL=0
MOVL C00794 V=800.0 PL=0
MOVL C00795 V=800.0 PL=0
MOVL C00796 V=800.0 PL=0
MOVL C00797 V=800.0 PL=0
MOVL C00798 V=800.0 PL=0
MOVL C00799 V=800.0 PL=0
MOVL C00800 V=800.0 PL=0
MOVL C00801 V=800.0 PL=0
MOVL C00802 V=800.0 PL=0
MOVL C00803 V=800.0 PL=0
MOVL C00804 V=800.0 PL=0
MOVL C00805 V=800.0 PL=0
MOVL C00806 V=800.0 PL=0
MOVL C00807 V=800.0 PL=0
MOVL C00808 V=800.0 PL=0
MOVL C00809 V=800.0 PL=0
MOVL C00810 V=800.0 PL=0
MOVL C00811 V=800.0 PL=0
MOVL C00812 V=800.0 PL=0
MOVL C00813 V=800.0 PL=0
MOVL C00814 V=800.0 PL=0
MOVL C00815 V=800.0 PL=0
MOVL C00816 V=800.0 PL=0
MOVL C00817 V=800.0 PL=0
MOVL C00818 V=800.0 PL=0
MOVL C00819 V=800.0 PL=0
MOVL C00820 V=800.0 PL=0
MOVL C00821 V=800.0 PL=0
MOVL C00822 V=800.0 PL=0
MOVL C00823 V=800.0 PL=0
MOVL C00824 V=800.0 PL=0
MOVL C00825 V=800.0 PL=0
MOVL C00826 V=800.0 PL=0
MOVL C00827 V=800.0 PL=0
MOVL C00828 V=800.0 PL=0
MOVL C00829 V=800.0 PL=0
MOVL C00830 V=800.0 PL=0
MOVL C00831 V=800.0 PL=0
MOVL C00832 V=800.0 PL=0
MOVL C00833 V=800.0 PL=0
MOVL C00834 V=800.0 PL=0
MOVL C00835 V=800.0 PL=0
MOVL C00836 V=800.0 PL=0
MOVL C00837 V=800.0 PL=0
MOVL C00838 V=800.0 PL=0
MOVL C00839 V=800.0 PL=0
MOVL C00840 V=800.0 PL=0
MOVL C00841 V=800.0 PL=0
MOVL C00842 V=800.0 PL=0
MOVL C00843 V=800.0 PL=0
MOVL C00844 V=800.0 PL=0
MOVL C00845 V=800.0 PL=0
MOVL C00846 V=800.0 PL=0
MOVL C00847 V=800.0 PL=0
MOVL C00848 V=800.0 PL=0
MOVL C00849 V=800.0 PL=0
MOVL C00850 V=800.0 PL=0
MOVL C00851 V=800.0 PL=0
MOVL C00852 V=800.0 PL=0
MOVL C00853 V=800.0 PL=0
MOVL C00854 V=800.0 PL=0
MOVL C00855 V=800.0 PL=0
MOVL C00856 V=800.0 PL=0
MOVL C00857 V=800.0 PL=0
MOVL C00858 V=800.0 PL=0
MOVL C00859 V=800.0 PL=0
MOVL C00860 V=800.0 PL=0
MOVL C00861 V=800.0 PL=0
MOVL C00862 V=800.0 PL=0
MOVL C00863 V=800.0 PL=0
MOVL C00864 V=800.0 PL=0
MOVL C00865 V=800.0 PL=0
MOVL C00866 V=800.0 PL=0
MOVL C00867 V=800.0 PL=0
MOVL C00868 V=800.0 PL=0
MOVL C00869 V=800.0 PL=0
MOVL C00870 V=800.0 PL=0
MOVL C00871 V=800.0 PL=0
MOVL C00872 V=800.0 PL=0
MOVL C00873 V=800.0 PL=0
MOVL C00874 V=800.0 PL=0
MOVL C00875 V=800.0 PL=0
MOVL C00876 V=800.0 PL=0
MOVL C00877 V=800.0 PL=0
MOVL C00878 V=800.0 PL=0
MOVL C00879 V=800.0 PL=0
MOVL C00880 V=800.0 PL=0
MOVL C00881 V=800.0 PL=0
MOVL C00882 V=800.0 PL=0
MOVL C00883 V=800.0 PL=0
MOVL C00884 V=800.0 PL=0
MOVL C00885 V=800.0 PL=0
MOVL C00886 V=800.0 PL=0
MOVL C00887 V=800.0 PL=0
MOVL C00888 V=800.0 PL=0
MOVL C00889 V=800.0 PL=0
MOVL C00890 V=800.0 PL=0
MOVL C00891 V=800.0 PL=0
MOVL C00892 V=800.0 PL=0
MOVL C00893 V=800.0 PL=0
MOVL C00894 V=800.0 PL=0
MOVL C00895 V=800.0 PL=0
MOVL C00896 V=800.0 PL=0
MOVL C00897 V=800.0 PL=0
MOVL C00898 V=800.0 PL=0
MOVL C00899 V=800.0 PL=0
MOVL C00900 V=800.0 PL=0
MOVL C00901 V=800.0 PL=0
MOVL C00902 V=800.0 PL=0
MOVL C00903 V=800.0 PL=0
MOVL C00904 V=800.0 PL=0
MOVL C00905 V=800.0 PL=0
MOVL C00906 V=800.0 PL=0
MOVL C00907 V=800.0 PL=0
MOVL C00908 V=800.0 PL=0
MOVL C00909 V=800.0 PL=0
MOVL C00910 V=800.0 PL=0
MOVL C00911 V=800.0 PL=0
MOVL C00912 V=800.0 PL=0
MOVL C00913 V=800.0 PL=0
MOVL C00914 V=800.0 PL=0
MOVL C00915 V=800.0 PL=0
MOVL C00916 V=800.0 PL=0
MOVL C00917 V=800.0 PL=0
MOVL C00918 V=800.0 PL=0
MOVL C00919 V=800.0 PL=0
MOVL C00920 V=800.0 PL=0
MOVL C00921 V=800.0 PL=0
MOVL C00922 V=800.0 PL=0
MOVL C00923 V=800.0 PL=0
MOVL C00924 V=800.0 PL=0
MOVL C00925 V=800.0 PL=0
MOVL C00926 V=800.0 PL=0
MOVL C00927 V=800.0 PL=0
MOVL C00928 V=800.0 PL=0
MOVL C00929 V=800.0 PL=0
MOVL C00930 V=800.0 PL=0
MOVL C00931 V=800.0 PL=0
MOVL C00932 V=800.0 PL=0
MOVL C00933 V=800.0 PL=0
MOVL C00934 V=800.0 PL=0
MOVL C00935 V=800.0 PL=0
MOVL C00936 V=800.0 PL=0
MOVL C00937 V=800.0 PL=0
MOVL C00938 V=800.0 PL=0
MOVL C00939 V=800.0 PL=0
MOVL C00940 V=800.0 PL=0
MOVL C00941 V=800.0 PL=0
MOVL C00942 V=800.0 PL=0
MOVL C00943 V=800.0 PL=0
MOVL C00944 V=800.0 PL=0
MOVL C00945 V=800.0 PL=0
MOVL C00946 V=800.0 PL=0
MOVL C00947 V=800.0 PL=0
MOVL C00948 V=800.0 PL=0
MOVL C00949 V=800.0 PL=0
MOVL C00950 V=800.0 PL=0
MOVL C00951 V=800.0 PL=0
MOVL C00952 V=800.0 PL=0
MOVL C00953 V=800.0 PL=0
MOVL C00954 V=800.0 PL=0
MOVL C00955 V=800.0 PL=0
MOVL C00956 V=800.0 PL=0
MOVL C00957 V=800.0 PL=0
MOVL C00958 V=800.0 PL=0
MOVL C00959 V=800.0 PL=0
MOVL C00960 V=800.0 PL=0
MOVL C00961 V=800.0 PL=0
MOVL C00962 V=800.0 PL=0
MOVL C00963 V=800.0 PL=0
MOVL C00964 V=800.0 PL=0
MOVL C00965 V=800.0 PL=0
MOVL C00966 V=800.0 PL=0
MOVL C00967 V=800.0 PL=0
MOVL C00968 V=800.0 PL=0
MOVL C00969 V=800.0 PL=0
MOVL C00970 V=800.0 PL=0
MOVL C00971 V=800.0 PL=0
MOVL C00972 V=800.0 PL=0
MOVL C00973 V=800.0 PL=0
MOVL C00974 V=800.0 PL=0
MOVL C00975 V=800.0 PL=0
MOVL C00976 V=800.0 PL=0
MOVL C00977 V=800.0 PL=0
MOVL C00978 V=800.0 PL=0
MOVL C00979 V=800.0 PL=0
MOVL C00980 V=800.0 PL=0
MOVL C00981 V=800.0 PL=0
MOVL C00982 V=800.0 PL=0
MOVL C00983 V=800.0 PL=0
MOVL C00984 V=800.0 PL=0
MOVL C00985 V=800.0 PL=0
MOVL C00986 V=800.0 PL=0
MOVL C00987 V=800.0 PL=0
MOVL C00988 V=800.0 PL=0
MOVL C00989 V=800.0 PL=0
MOVL C00990 V=800.0 PL=0
MOVL C00991 V=800.0 PL=0
MOVL C00992 V=800.0 PL=0
MOVL C00993 V=800.0 PL=0
MOVL C00994 V=800.0 PL=0
MOVL C00995 V=800.0 PL=0
MOVL C00996 V=800.0 PL=0
MOVL C00997 V=800.0 PL=0
MOVL C00998 V=800.0 PL=0
MOVL C00999 V=800.0 PL=0
MOVL C01000 V=800.0 PL=0
MOVL C01001 V=800.0 PL=0
MOVL C01002 V=800.0 PL=0
MOVL C01003 V=800.0 PL=0
MOVL C01004 V=800.0 PL=0
MOVL C01005 V=800.0 PL=0
MOVL C01006 V=800.0 PL=0
MOVL C01007 V=800.0 PL=0
MOVL C01008 V=800.0 PL=0
MOVL C01009 V=800.0 PL=0
MOVL C01010 V=800.0 PL=0
MOVL C01011 V=800.0 PL=0
MOVL C01012 V=800.0 PL=0
MOVL C01013 V=800.0 PL=0
MOVL C01014 V=800.0 PL=0
MOVL C01015 V=800.0 PL=0
MOVL C01016 V=800.0 PL=0
MOVL C01017 V=800.0 PL=0
MOVL C01018 V=800.0 PL=0
MOVL C01019 V=800.0 PL=0
MOVL C01020 V=800.0 PL=0
MOVL C01021 V=800.0 PL=0
MOVL C01022 V=800.0 PL=0
MOVL C01023 V=800.0 PL=0
MOVL C01024 V=800.0 PL=0
MOVL C01025 V=800.0 PL=0
MOVL C01026 V=800.0 PL=0
MOVL C01027 V=800.0 PL=0
MOVL C01028 V=800.0 PL=0
MOVL C01029 V=800.0 PL=0
MOVL C01030 V=800.0 PL=0
MOVL C01031 V=800.0 PL=0
MOVL C01032 V=800.0 PL=0
MOVL C01033 V=800.0 PL=0
MOVL C01034 V=800.0 PL=0
MOVL C01035 V=800.0 PL=0
MOVL C01036 V=800.0 PL=0
MOVL C01037 V=800.0 PL=0
MOVL C01038 V=800.0 PL=0
MOVL C01039 V=800.0 PL=0
MOVL C01040 V=800.0 PL=0
MOVL C01041 V=800.0 PL=0
MOVL C01042 V=800.0 PL=0
MOVL C01043 V=800.0 PL=0
MOVL C01044 V=800.0 PL=0
MOVL C01045 V=800.0 PL=0
MOVL C01046 V=800.0 PL=0
MOVL C01047 V=800.0 PL=0
MOVL C01048 V=800.0 PL=0
MOVL C01049 V=800.0 PL=0
MOVL C01050 V=800.0 PL=0
MOVL C01051 V=800.0 PL=0
MOVL C01052 V=800.0 PL=0
MOVL C01053 V=800.0 PL=0
MOVL C01054 V=800.0 PL=0
MOVL C01055 V=800.0 PL=0
MOVL C01056 V=800.0 PL=0
MOVL C01057 V=800.0 PL=0
MOVL C01058 V=800.0 PL=0
MOVL C01059 V=800.0 PL=0
MOVL C01060 V=800.0 PL=0
MOVL C01061 V=800.0 PL=0
MOVL C01062 V=800.0 PL=0
MOVL C01063 V=800.0 PL=0
MOVL C01064 V=800.0 PL=0
MOVL C01065 V=800.0 PL=0
MOVL C01066 V=800.0 PL=0
MOVL C01067 V=800.0 PL=0
MOVL C01068 V=800.0 PL=0
MOVL C01069 V=800.0 PL=0
MOVL C01070 V=800.0 PL=0
MOVL C01071 V=800.0 PL=0
MOVL C01072 V=800.0 PL=0
MOVL C01073 V=800.0 PL=0
MOVL C01074 V=800.0 PL=0
MOVL C01075 V=800.0 PL=0
MOVL C01076 V=800.0 PL=0
MOVL C01077 V=800.0 PL=0
MOVL C01078 V=800.0 PL=0
MOVL C01079 V=800.0 PL=0
MOVL C01080 V=800.0 PL=0
MOVL C01081 V=800.0 PL=0
MOVL C01082 V=800.0 PL=0
MOVL C01083 V=800.0 PL=0
MOVL C01084 V=800.0 PL=0
MOVL C01085 V=800.0 PL=0
MOVL C01086 V=800.0 PL=0
MOVL C01087 V=800.0 PL=0
MOVL C01088 V=800.0 PL=0
MOVL C01089 V=800.0 PL=0
MOVL C01090 V=800.0 PL=0
MOVL C01091 V=800.0 PL=0
MOVL C01092 V=800.0 PL=0
MOVL C01093 V=800.0 PL=0
MOVL C01094 V=800.0 PL=0
MOVL C01095 V=800.0 PL=0
MOVL C01096 V=800.0 PL=0
MOVL C01097 V=800.0 PL=0
MOVL C01098 V=800.0 PL=0
MOVL C01099 V=800.0 PL=0
MOVL C01100 V=800.0 PL=0
MOVL C01101 V=800.0 PL=0
MOVL C01102 V=800.0 PL=0
MOVL C01103 V=800.0 PL=0
MOVL C01104 V=800.0 PL=0
MOVL C01105 V=800.0 PL=0
MOVL C01106 V=800.0 PL=0
MOVL C01107 V=800.0 PL=0
MOVL C01108 V=800.0 PL=0
MOVL C01109 V=800.0 PL=0
MOVL C01110 V=800.0 PL=0
MOVL C01111 V=800.0 PL=0
MOVL C01112 V=800.0 PL=0
MOVL C01113 V=800.0 PL=0
MOVL C01114 V=800.0 PL=0
MOVL C01115 V=800.0 PL=0
MOVL C01116 V=800.0 PL=0
MOVL C01117 V=800.0 PL=0
MOVL C01118 V=800.0 PL=0
MOVL C01119 V=800.0 PL=0
MOVL C01120 V=800.0 PL=0
MOVL C01121 V=800.0 PL=0
MOVL C01122 V=800.0 PL=0
MOVL C01123 V=800.0 PL=0
MOVL C01124 V=800.0 PL=0
MOVL C01125 V=800.0 PL=0
MOVL C01126 V=800.0 PL=0
MOVL C01127 V=800.0 PL=0
MOVL C01128 V=800.0 PL=0
MOVL C01129 V=800.0 PL=0
MOVL C01130 V=800.0 PL=0
MOVL C01131 V=800.0 PL=0
MOVL C01132 V=800.0 PL=0
MOVL C01133 V=800.0 PL=0
MOVL C01134 V=800.0 PL=0
MOVL C01135 V=800.0 PL=0
MOVL C01136 V=800.0 PL=0
MOVL C01137 V=800.0 PL=0
MOVL C01138 V=800.0 PL=0
MOVL C01139 V=800.0 PL=0
MOVL C01140 V=800.0 PL=0
MOVL C01141 V=800.0 PL=0
MOVL C01142 V=800.0 PL=0
MOVL C01143 V=800.0 PL=0
MOVL C01144 V=800.0 PL=0
MOVL C01145 V=800.0 PL=0
MOVL C01146 V=800.0 PL=0
MOVL C01147 V=800.0 PL=0
MOVL C01148 V=800.0 PL=0
MOVL C01149 V=800.0 PL=0
MOVL C01150 V=800.0 PL=0
MOVL C01151 V=800.0 PL=0
MOVL C01152 V=800.0 PL=0
MOVL C01153 V=800.0 PL=0
MOVL C01154 V=800.0 PL=0
MOVL C01155 V=800.0 PL=0
MOVL C01156 V=800.0 PL=0
MOVL C01157 V=800.0 PL=0
MOVL C01158 V=800.0 PL=0
MOVL C01159 V=800.0 PL=0
MOVL C01160 V=800.0 PL=0
MOVL C01161 V=800.0 PL=0
MOVL C01162 V=800.0 PL=0
MOVL C01163 V=800.0 PL=0
MOVL C01164 V=800.0 PL=0
MOVL C01165 V=800.0 PL=0
MOVL C01166 V=800.0 PL=0
MOVL C01167 V=800.0 PL=0
MOVL C01168 V=800.0 PL=0
MOVL C01169 V=800.0 PL=0
MOVL C01170 V=800.0 PL=0
MOVL C01171 V=800.0 PL=0
MOVL C01172 V=800.0 PL=0
MOVL C01173 V=800.0 PL=0
MOVL C01174 V=800.0 PL=0
MOVL C01175 V=800.0 PL=0
MOVL C01176 V=800.0 PL=0
MOVL C01177 V=800.0 PL=0
MOVL C01178 V=800.0 PL=0
MOVL C01179 V=800.0 PL=0
MOVL C01180 V=800.0 PL=0
MOVL C01181 V=800.0 PL=0
MOVL C01182 V=800.0 PL=0
MOVL C01183 V=800.0 PL=0
MOVL C01184 V=800.0 PL=0
MOVL C01185 V=800.0 PL=0
MOVL C01186 V=800.0 PL=0
MOVL C01187 V=800.0 PL=0
MOVL C01188 V=800.0 PL=0
MOVL C01189 V=800.0 PL=0
MOVL C01190 V=800.0 PL=0
MOVL C01191 V=800.0 PL=0
MOVL C01192 V=800.0 PL=0
MOVL C01193 V=800.0 PL=0
MOVL C01194 V=800.0 PL=0
MOVL C01195 V=800.0 PL=0
MOVL C01196 V=800.0 PL=0
MOVL C01197 V=800.0 PL=0
MOVL C01198 V=800.0 PL=0
MOVL C01199 V=800.0 PL=0
MOVL C01200 V=800.0 PL=0
MOVL C01201 V=800.0 PL=0
MOVL C01202 V=800.0 PL=0
MOVL C01203 V=800.0 PL=0
MOVL C01204 V=800.0 PL=0
MOVL C01205 V=800.0 PL=0
MOVL C01206 V=800.0 PL=0
MOVL C01207 V=800.0 PL=0
MOVL C01208 V=800.0 PL=0
MOVL C01209 V=800.0 PL=0
MOVL C01210 V=800.0 PL=0
MOVL C01211 V=800.0 PL=0
MOVL C01212 V=800.0 PL=0
MOVL C01213 V=800.0 PL=0
MOVL C01214 V=800.0 PL=0
MOVL C01215 V=800.0 PL=0
MOVL C01216 V=800.0 PL=0
MOVL C01217 V=800.0 PL=0
MOVL C01218 V=800.0 PL=0
MOVL C01219 V=800.0 PL=0
MOVL C01220 V=800.0 PL=0
MOVL C01221 V=800.0 PL=0
MOVL C01222 V=800.0 PL=0
MOVL C01223 V=800.0 PL=0
MOVL C01224 V=800.0 PL=0
MOVL C01225 V=800.0 PL=0
MOVL C01226 V=800.0 PL=0
MOVL C01227 V=800.0 PL=0
MOVL C01228 V=800.0 PL=0
MOVL C01229 V=800.0 PL=0
MOVL C01230 V=800.0 PL=0
MOVL C01231 V=800.0 PL=0
MOVL C01232 V=800.0 PL=0
MOVL C01233 V=800.0 PL=0
MOVL C01234 V=800.0 PL=0
MOVL C01235 V=800.0 PL=0
MOVL C01236 V=800.0 PL=0
MOVL C01237 V=800.0 PL=0
MOVL C01238 V=800.0 PL=0
MOVL C01239 V=800.0 PL=0
MOVL C01240 V=800.0 PL=0
MOVL C01241 V=800.0 PL=0
MOVL C01242 V=800.0 PL=0
MOVL C01243 V=800.0 PL=0
MOVL C01244 V=800.0 PL=0
MOVL C01245 V=800.0 PL=0
MOVL C01246 V=800.0 PL=0
MOVL C01247 V=800.0 PL=0
MOVL C01248 V=800.0 PL=0
MOVL C01249 V=800.0 PL=0
MOVL C01250 V=800.0 PL=0
MOVL C01251 V=800.0 PL=0
MOVL C01252 V=800.0 PL=0
MOVL C01253 V=800.0 PL=0
MOVL C01254 V=800.0 PL=0
MOVL C01255 V=800.0 PL=0
MOVL C01256 V=800.0 PL=0
MOVL C01257 V=800.0 PL=0
MOVL C01258 V=800.0 PL=0
MOVL C01259 V=800.0 PL=0
MOVL C01260 V=800.0 PL=0
MOVL C01261 V=800.0 PL=0
MOVL C01262 V=800.0 PL=0
MOVL C01263 V=800.0 PL=0
MOVL C01264 V=800.0 PL=0
MOVL C01265 V=800.0 PL=0
MOVL C01266 V=800.0 PL=0
MOVL C01267 V=800.0 PL=0
MOVL C01268 V=800.0 PL=0
MOVL C01269 V=800.0 PL=0
MOVL C01270 V=800.0 PL=0
MOVL C01271 V=800.0 PL=0
MOVL C01272 V=800.0 PL=0
MOVL C01273 V=800.0 PL=0
MOVL C01274 V=800.0 PL=0
MOVL C01275 V=800.0 PL=0
MOVL C01276 V=800.0 PL=0
MOVL C01277 V=800.0 PL=0
MOVL C01278 V=800.0 PL=0
MOVL C01279 V=800.0 PL=0
MOVL C01280 V=800.0 PL=0
MOVL C01281 V=800.0 PL=0
MOVL C01282 V=800.0 PL=0
MOVL C01283 V=800.0 PL=0
MOVL C01284 V=800.0 PL=0
MOVL C01285 V=800.0 PL=0
MOVL C01286 V=800.0 PL=0
MOVL C01287 V=800.0 PL=0
MOVL C01288 V=800.0 PL=0
MOVL C01289 V=800.0 PL=0
MOVL C01290 V=800.0 PL=0
MOVL C01291 V=800.0 PL=0
MOVL C01292 V=800.0 PL=0
MOVL C01293 V=800.0 PL=0
MOVL C01294 V=800.0 PL=0
MOVL C01295 V=800.0 PL=0
MOVL C01296 V=800.0 PL=0
MOVL C01297 V=800.0 PL=0
MOVL C01298 V=800.0 PL=0
MOVL C01299 V=800.0 PL=0
MOVL C01300 V=800.0 PL=0
MOVL C01301 V=800.0 PL=0
MOVL C01302 V=800.0 PL=0
MOVL C01303 V=800.0 PL=0
MOVL C01304 V=800.0 PL=0
MOVL C01305 V=800.0 PL=0
MOVL C01306 V=800.0 PL=0
MOVL C01307 V=800.0 PL=0
MOVL C01308 V=800.0 PL=0
MOVL C01309 V=800.0 PL=0
MOVL C01310 V=800.0 PL=0
MOVL C01311 V=800.0 PL=0
MOVL C01312 V=800.0 PL=0
MOVL C01313 V=800.0 PL=0
MOVL C01314 V=800.0 PL=0
MOVL C01315 V=800.0 PL=0
MOVL C01316 V=800.0 PL=0
MOVL C01317 V=800.0 PL=0
MOVL C01318 V=800.0 PL=0
MOVL C01319 V=800.0 PL=0
MOVL C01320 V=800.0 PL=0
MOVL C01321 V=800.0 PL=0
MOVL C01322 V=800.0 PL=0
MOVL C01323 V=800.0 PL=0
MOVL C01324 V=800.0 PL=0
MOVL C01325 V=800.0 PL=0
MOVL C01326 V=800.0 PL=0
MOVL C01327 V=800.0 PL=0
MOVL C01328 V=800.0 PL=0
MOVL C01329 V=800.0 PL=0
MOVL C01330 V=800.0 PL=0
MOVL C01331 V=800.0 PL=0
MOVL C01332 V=800.0 PL=0
MOVL C01333 V=800.0 PL=0
MOVL C01334 V=800.0 PL=0
MOVL C01335 V=800.0 PL=0
MOVL C01336 V=800.0 PL=0
MOVL C01337 V=800.0 PL=0
MOVL C01338 V=800.0 PL=0
MOVL C01339 V=800.0 PL=0
MOVL C01340 V=800.0 PL=0
MOVL C01341 V=800.0 PL=0
MOVL C01342 V=800.0 PL=0
MOVL C01343 V=800.0 PL=0
MOVL C01344 V=800.0 PL=0
MOVL C01345 V=800.0 PL=0
MOVL C01346 V=800.0 PL=0
MOVL C01347 V=800.0 PL=0
MOVL C01348 V=800.0 PL=0
MOVL C01349 V=800.0 PL=0
MOVL C01350 V=800.0 PL=0
MOVL C01351 V=800.0 PL=0
MOVL C01352 V=800.0 PL=0
MOVL C01353 V=800.0 PL=0
MOVL C01354 V=800.0 PL=0
MOVL C01355 V=800.0 PL=0
MOVL C01356 V=800.0 PL=0
MOVL C01357 V=800.0 PL=0
MOVL C01358 V=800.0 PL=0
MOVL C01359 V=800.0 PL=0
MOVL C01360 V=800.0 PL=0
MOVL C01361 V=800.0 PL=0
MOVL C01362 V=800.0 PL=0
MOVL C01363 V=800.0 PL=0
MOVL C01364 V=800.0 PL=0
MOVL C01365 V=800.0 PL=0
MOVL C01366 V=800.0 PL=0
MOVL C01367 V=800.0 PL=0
MOVL C01368 V=800.0 PL=0
MOVL C01369 V=800.0 PL=0
MOVL C01370 V=800.0 PL=0
MOVL C01371 V=800.0 PL=0
MOVL C01372 V=800.0 PL=0
MOVL C01373 V=800.0 PL=0
MOVL C01374 V=800.0 PL=0
MOVL C01375 V=800.0 PL=0
MOVL C01376 V=800.0 PL=0
MOVL C01377 V=800.0 PL=0
MOVL C01378 V=800.0 PL=0
MOVL C01379 V=800.0 PL=0
MOVL C01380 V=800.0 PL=0
MOVL C01381 V=800.0 PL=0
MOVL C01382 V=800.0 PL=0
MOVL C01383 V=800.0 PL=0
MOVL C01384 V=800.0 PL=0
MOVL C01385 V=800.0 PL=0
MOVL C01386 V=800.0 PL=0
MOVL C01387 V=800.0 PL=0
MOVL C01388 V=800.0 PL=0
MOVL C01389 V=800.0 PL=0
MOVL C01390 V=800.0 PL=0
MOVL C01391 V=800.0 PL=0
MOVL C01392 V=800.0 PL=0
MOVL C01393 V=800.0 PL=0
MOVL C01394 V=800.0 PL=0
MOVL C01395 V=800.0 PL=0
MOVL C01396 V=800.0 PL=0
MOVL C01397 V=800.0 PL=0
MOVL C01398 V=800.0 PL=0
MOVL C01399 V=800.0 PL=0
MOVL C01400 V=800.0 PL=0
MOVL C01401 V=800.0 PL=0
MOVL C01402 V=800.0 PL=0
MOVL C01403 V=800.0 PL=0
MOVL C01404 V=800.0 PL=0
MOVL C01405 V=800.0 PL=0
MOVL C01406 V=800.0 PL=0
MOVL C01407 V=800.0 PL=0
MOVL C01408 V=800.0 PL=0
MOVL C01409 V=800.0 PL=0
MOVL C01410 V=800.0 PL=0
MOVL C01411 V=800.0 PL=0
MOVL C01412 V=800.0 PL=0
MOVL C01413 V=800.0 PL=0
MOVL C01414 V=800.0 PL=0
MOVL C01415 V=800.0 PL=0
MOVL C01416 V=800.0 PL=0
MOVL C01417 V=800.0 PL=0
MOVL C01418 V=800.0 PL=0
MOVL C01419 V=800.0 PL=0
MOVL C01420 V=800.0 PL=0
MOVL C01421 V=800.0 PL=0
MOVL C01422 V=800.0 PL=0
MOVL C01423 V=800.0 PL=0
MOVL C01424 V=800.0 PL=0
MOVL C01425 V=800.0 PL=0
MOVL C01426 V=800.0 PL=0
MOVL C01427 V=800.0 PL=0
MOVL C01428 V=800.0 PL=0
MOVL C01429 V=800.0 PL=0
MOVL C01430 V=800.0 PL=0
MOVL C01431 V=800.0 PL=0
MOVL C01432 V=800.0 PL=0
MOVL C01433 V=800.0 PL=0
MOVL C01434 V=800.0 PL=0
MOVL C01435 V=800.0 PL=0
MOVL C01436 V=800.0 PL=0
MOVL C01437 V=800.0 PL=0
MOVL C01438 V=800.0 PL=0
MOVL C01439 V=800.0 PL=0
MOVL C01440 V=800.0 PL=0
MOVL C01441 V=800.0 PL=0
MOVL C01442 V=800.0 PL=0
MOVL C01443 V=800.0 PL=0
MOVL C01444 V=800.0 PL=0
MOVL C01445 V=800.0 PL=0
MOVL C01446 V=800.0 PL=0
MOVL C01447 V=800.0 PL=0
MOVL C01448 V=800.0 PL=0
MOVL C01449 V=800.0 PL=0
MOVL C01450 V=800.0 PL=0
MOVL C01451 V=800.0 PL=0
MOVL C01452 V=800.0 PL=0
MOVL C01453 V=800.0 PL=0
MOVL C01454 V=800.0 PL=0
MOVL C01455 V=800.0 PL=0
MOVL C01456 V=800.0 PL=0
MOVL C01457 V=800.0 PL=0
MOVL C01458 V=800.0 PL=0
MOVL C01459 V=800.0 PL=0
MOVL C01460 V=800.0 PL=0
MOVL C01461 V=800.0 PL=0
MOVL C01462 V=800.0 PL=0
MOVL C01463 V=800.0 PL=0
MOVL C01464 V=800.0 PL=0
MOVL C01465 V=800.0 PL=0
MOVL C01466 V=800.0 PL=0
MOVL C01467 V=800.0 PL=0
MOVL C01468 V=800.0 PL=0
MOVL C01469 V=800.0 PL=0
MOVL C01470 V=800.0 PL=0
MOVL C01471 V=800.0 PL=0
MOVL C01472 V=800.0 PL=0
MOVL C01473 V=800.0 PL=0
MOVL C01474 V=800.0 PL=0
MOVL C01475 V=800.0 PL=0
MOVL C01476 V=800.0 PL=0
MOVL C01477 V=800.0 PL=0
MOVL C01478 V=800.0 PL=0
MOVL C01479 V=800.0 PL=0
MOVL C01480 V=800.0 PL=0
MOVL C01481 V=800.0 PL=0
MOVL C01482 V=800.0 PL=0
MOVL C01483 V=800.0 PL=0
MOVL C01484 V=800.0 PL=0
MOVL C01485 V=800.0 PL=0
MOVL C01486 V=800.0 PL=0
MOVL C01487 V=800.0 PL=0
MOVL C01488 V=800.0 PL=0
MOVL C01489 V=800.0 PL=0
MOVL C01490 V=800.0 PL=0
MOVL C01491 V=800.0 PL=0
MOVL C01492 V=800.0 PL=0
MOVL C01493 V=800.0 PL=0
MOVL C01494 V=800.0 PL=0
MOVL C01495 V=800.0 PL=0
MOVL C01496 V=800.0 PL=0
MOVL C01497 V=800.0 PL=0
MOVL C01498 V=800.0 PL=0
MOVL C01499 V=800.0 PL=0
MOVL C01500 V=800.0 PL=0
MOVL C01501 V=800.0 PL=0
MOVL C01502 V=800.0 PL=0
MOVL C01503 V=800.0 PL=0
MOVL C01504 V=800.0 PL=0
MOVL C01505 V=800.0 PL=0
MOVL C01506 V=800.0 PL=0
MOVL C01507 V=800.0 PL=0
MOVL C01508 V=800.0 PL=0
MOVL C01509 V=800.0 PL=0
MOVL C01510 V=800.0 PL=0
MOVL C01511 V=800.0 PL=0
MOVL C01512 V=800.0 PL=0
MOVL C01513 V=800.0 PL=0
MOVL C01514 V=800.0 PL=0
MOVL C01515 V=800.0 PL=0
MOVL C01516 V=800.0 PL=0
MOVL C01517 V=800.0 PL=0
MOVL C01518 V=800.0 PL=0
MOVL C01519 V=800.0 PL=0
MOVL C01520 V=800.0 PL=0
MOVL C01521 V=800.0 PL=0
MOVL C01522 V=800.0 PL=0
MOVL C01523 V=800.0 PL=0
MOVL C01524 V=800.0 PL=0
MOVL C01525 V=800.0 PL=0
MOVL C01526 V=800.0 PL=0
MOVL C01527 V=800.0 PL=0
MOVL C01528 V=800.0 PL=0
MOVL C01529 V=800.0 PL=0
MOVL C01530 V=800.0 PL=0
MOVL C01531 V=800.0 PL=0
MOVL C01532 V=800.0 PL=0
MOVL C01533 V=800.0 PL=0
MOVL C01534 V=800.0 PL=0
MOVL C01535 V=800.0 PL=0
MOVL C01536 V=800.0 PL=0
MOVL C01537 V=800.0 PL=0
MOVL C01538 V=800.0 PL=0
MOVL C01539 V=800.0 PL=0
MOVL C01540 V=800.0 PL=0
MOVL C01541 V=800.0 PL=0
MOVL C01542 V=800.0 PL=0
MOVL C01543 V=800.0 PL=0
MOVL C01544 V=800.0 PL=0
MOVL C01545 V=800.0 PL=0
MOVL C01546 V=800.0 PL=0
MOVL C01547 V=800.0 PL=0
MOVL C01548 V=800.0 PL=0
MOVL C01549 V=800.0 PL=0
MOVL C01550 V=800.0 PL=0
MOVL C01551 V=800.0 PL=0
MOVL C01552 V=800.0 PL=0
MOVL C01553 V=800.0 PL=0
MOVL C01554 V=800.0 PL=0
MOVL C01555 V=800.0 PL=0
MOVL C01556 V=800.0 PL=0
MOVL C01557 V=800.0 PL=0
MOVL C01558 V=800.0 PL=0
MOVL C01559 V=800.0 PL=0
MOVL C01560 V=800.0 PL=0
MOVL C01561 V=800.0 PL=0
MOVL C01562 V=800.0 PL=0
MOVL C01563 V=800.0 PL=0
MOVL C01564 V=800.0 PL=0
MOVL C01565 V=800.0 PL=0
MOVL C01566 V=800.0 PL=0
MOVL C01567 V=800.0 PL=0
MOVL C01568 V=800.0 PL=0
MOVL C01569 V=800.0 PL=0
MOVL C01570 V=800.0 PL=0
MOVL C01571 V=800.0 PL=0
MOVL C01572 V=800.0 PL=0
MOVL C01573 V=800.0 PL=0
MOVL C01574 V=800.0 PL=0
MOVL C01575 V=800.0 PL=0
MOVL C01576 V=800.0 PL=0
MOVL C01577 V=800.0 PL=0
MOVL C01578 V=800.0 PL=0
MOVL C01579 V=800.0 PL=0
MOVL C01580 V=800.0 PL=0
MOVL C01581 V=800.0 PL=0
MOVL C01582 V=800.0 PL=0
MOVL C01583 V=800.0 PL=0
MOVL C01584 V=800.0 PL=0
MOVL C01585 V=800.0 PL=0
MOVL C01586 V=800.0 PL=0
MOVL C01587 V=800.0 PL=0
MOVL C01588 V=800.0 PL=0
MOVL C01589 V=800.0 PL=0
MOVL C01590 V=800.0 PL=0
MOVL C01591 V=800.0 PL=0
MOVL C01592 V=800.0 PL=0
MOVL C01593 V=800.0 PL=0
MOVL C01594 V=800.0 PL=0
MOVL C01595 V=800.0 PL=0
MOVL C01596 V=800.0 PL=0
MOVL C01597 V=800.0 PL=0
MOVL C01598 V=800.0 PL=0
MOVL C01599 V=800.0 PL=0
MOVL C01600 V=800.0 PL=0
MOVL C01601 V=800.0 PL=0
MOVL C01602 V=800.0 PL=0
MOVL C01603 V=800.0 PL=0
MOVL C01604 V=800.0 PL=0
MOVL C01605 V=800.0 PL=0
MOVL C01606 V=800.0 PL=0
MOVL C01607 V=800.0 PL=0
MOVL C01608 V=800.0 PL=0
MOVL C01609 V=800.0 PL=0
MOVL C01610 V=800.0 PL=0
MOVL C01611 V=800.0 PL=0
MOVL C01612 V=800.0 PL=0
MOVL C01613 V=800.0 PL=0
MOVL C01614 V=800.0 PL=0
MOVL C01615 V=800.0 PL=0
MOVL C01616 V=800.0 PL=0
MOVL C01617 V=800.0 PL=0
MOVL C01618 V=800.0 PL=0
MOVL C01619 V=800.0 PL=0
MOVL C01620 V=800.0 PL=0
MOVL C01621 V=800.0 PL=0
MOVL C01622 V=800.0 PL=0
MOVL C01623 V=800.0 PL=0
MOVL C01624 V=800.0 PL=0
MOVL C01625 V=800.0 PL=0
MOVL C01626 V=800.0 PL=0
MOVL C01627 V=800.0 PL=0
MOVL C01628 V=800.0 PL=0
MOVL C01629 V=800.0 PL=0
MOVL C01630 V=800.0 PL=0
MOVL C01631 V=800.0 PL=0
MOVL C01632 V=800.0 PL=0
MOVL C01633 V=800.0 PL=0
MOVL C01634 V=800.0 PL=0
MOVL C01635 V=800.0 PL=0
MOVL C01636 V=800.0 PL=0
MOVL C01637 V=800.0 PL=0
MOVL C01638 V=800.0 PL=0
MOVL C01639 V=800.0 PL=0
MOVL C01640 V=800.0 PL=0
MOVL C01641 V=800.0 PL=0
MOVL C01642 V=800.0 PL=0
MOVL C01643 V=800.0 PL=0
MOVL C01644 V=800.0 PL=0
MOVL C01645 V=800.0 PL=0
MOVL C01646 V=800.0 PL=0
MOVL C01647 V=800.0 PL=0
MOVL C01648 V=800.0 PL=0
MOVL C01649 V=800.0 PL=0
MOVL C01650 V=800.0 PL=0
MOVL C01651 V=800.0 PL=0
MOVL C01652 V=800.0 PL=0
MOVL C01653 V=800.0 PL=0
MOVL C01654 V=800.0 PL=0
MOVL C01655 V=800.0 PL=0
MOVL C01656 V=800.0 PL=0
MOVL C01657 V=800.0 PL=0
MOVL C01658 V=800.0 PL=0
MOVL C01659 V=800.0 PL=0
MOVL C01660 V=800.0 PL=0
MOVL C01661 V=800.0 PL=0
MOVL C01662 V=800.0 PL=0
MOVL C01663 V=800.0 PL=0
MOVL C01664 V=800.0 PL=0
MOVL C01665 V=800.0 PL=0
MOVL C01666 V=800.0 PL=0
MOVL C01667 V=800.0 PL=0
MOVL C01668 V=800.0 PL=0
MOVL C01669 V=800.0 PL=0
MOVL C01670 V=800.0 PL=0
MOVL C01671 V=800.0 PL=0
MOVL C01672 V=800.0 PL=0
MOVL C01673 V=800.0 PL=0
MOVL C01674 V=800.0 PL=0
MOVL C01675 V=800.0 PL=0
MOVL C01676 V=800.0 PL=0
MOVL C01677 V=800.0 PL=0
MOVL C01678 V=800.0 PL=0
MOVL C01679 V=800.0 PL=0
MOVL C01680 V=800.0 PL=0
MOVL C01681 V=800.0 PL=0
MOVL C01682 V=800.0 PL=0
MOVL C01683 V=800.0 PL=0
MOVL C01684 V=800.0 PL=0
MOVL C01685 V=800.0 PL=0
MOVL C01686 V=800.0 PL=0
MOVL C01687 V=800.0 PL=0
MOVL C01688 V=800.0 PL=0
MOVL C01689 V=800.0 PL=0
MOVL C01690 V=800.0 PL=0
MOVL C01691 V=800.0 PL=0
MOVL C01692 V=800.0 PL=0
MOVL C01693 V=800.0 PL=0
MOVL C01694 V=800.0 PL=0
MOVL C01695 V=800.0 PL=0
MOVL C01696 V=800.0 PL=0
MOVL C01697 V=800.0 PL=0
MOVL C01698 V=800.0 PL=0
MOVL C01699 V=800.0 PL=0
MOVL C01700 V=800.0 PL=0
MOVL C01701 V=800.0 PL=0
MOVL C01702 V=800.0 PL=0
MOVL C01703 V=800.0 PL=0
MOVL C01704 V=800.0 PL=0
MOVL C01705 V=800.0 PL=0
MOVL C01706 V=800.0 PL=0
MOVL C01707 V=800.0 PL=0
MOVL C01708 V=800.0 PL=0
MOVL C01709 V=800.0 PL=0
MOVL C01710 V=800.0 PL=0
MOVL C01711 V=800.0 PL=0
MOVL C01712 V=800.0 PL=0
MOVL C01713 V=800.0 PL=0
MOVL C01714 V=800.0 PL=0
MOVL C01715 V=800.0 PL=0
MOVL C01716 V=800.0 PL=0
MOVL C01717 V=800.0 PL=0
MOVL C01718 V=800.0 PL=0
MOVL C01719 V=800.0 PL=0
MOVL C01720 V=800.0 PL=0
MOVL C01721 V=800.0 PL=0
MOVL C01722 V=800.0 PL=0
MOVL C01723 V=800.0 PL=0
MOVL C01724 V=800.0 PL=0
MOVL C01725 V=800.0 PL=0
MOVL C01726 V=800.0 PL=0
MOVL C01727 V=800.0 PL=0
MOVL C01728 V=800.0 PL=0
MOVL C01729 V=800.0 PL=0
MOVL C01730 V=800.0 PL=0
MOVL C01731 V=800.0 PL=0
MOVL C01732 V=800.0 PL=0
MOVL C01733 V=800.0 PL=0
MOVL C01734 V=800.0 PL=0
MOVL C01735 V=800.0 PL=0
MOVL C01736 V=800.0 PL=0
MOVL C01737 V=800.0 PL=0
MOVL C01738 V=800.0 PL=0
MOVL C01739 V=800.0 PL=0
MOVL C01740 V=800.0 PL=0
MOVL C01741 V=800.0 PL=0
MOVL C01742 V=800.0 PL=0
MOVL C01743 V=800.0 PL=0
MOVL C01744 V=800.0 PL=0
MOVL C01745 V=800.0 PL=0
MOVL C01746 V=800.0 PL=0
MOVL C01747 V=800.0 PL=0
MOVL C01748 V=800.0 PL=0
MOVL C01749 V=800.0 PL=0
MOVL C01750 V=800.0 PL=0
MOVL C01751 V=800.0 PL=0
MOVL C01752 V=800.0 PL=0
MOVL C01753 V=800.0 PL=0
MOVL C01754 V=800.0 PL=0
MOVL C01755 V=800.0 PL=0
MOVL C01756 V=800.0 PL=0
MOVL C01757 V=800.0 PL=0
MOVL C01758 V=800.0 PL=0
MOVL C01759 V=800.0 PL=0
MOVL C01760 V=800.0 PL=0
MOVL C01761 V=800.0 PL=0
MOVL C01762 V=800.0 PL=0
MOVL C01763 V=800.0 PL=0
MOVL C01764 V=800.0 PL=0
MOVL C01765 V=800.0 PL=0
MOVL C01766 V=800.0 PL=0
MOVL C01767 V=800.0 PL=0
MOVL C01768 V=800.0 PL=0
MOVL C01769 V=800.0 PL=0
MOVL C01770 V=800.0 PL=0
MOVL C01771 V=800.0 PL=0
MOVL C01772 V=800.0 PL=0
MOVL C01773 V=800.0 PL=0
MOVL C01774 V=800.0 PL=0
MOVL C01775 V=800.0 PL=0
MOVL C01776 V=800.0 PL=0
MOVL C01777 V=800.0 PL=0
MOVL C01778 V=800.0 PL=0
MOVL C01779 V=800.0 PL=0
MOVL C01780 V=800.0 PL=0
MOVL C01781 V=800.0 PL=0
MOVL C01782 V=800.0 PL=0
MOVL C01783 V=800.0 PL=0
MOVL C01784 V=800.0 PL=0
MOVL C01785 V=800.0 PL=0
MOVL C01786 V=800.0 PL=0
MOVL C01787 V=800.0 PL=0
MOVL C01788 V=800.0 PL=0
MOVL C01789 V=800.0 PL=0
MOVL C01790 V=800.0 PL=0
MOVL C01791 V=800.0 PL=0
MOVL C01792 V=800.0 PL=0
MOVL C01793 V=800.0 PL=0
MOVL C01794 V=800.0 PL=0
MOVL C01795 V=800.0 PL=0
MOVL C01796 V=800.0 PL=0
MOVL C01797 V=800.0 PL=0
MOVL C01798 V=800.0 PL=0
MOVL C01799 V=800.0 PL=0
MOVL C01800 V=800.0 PL=0
MOVL C01801 V=800.0 PL=0
MOVL C01802 V=800.0 PL=0
MOVL C01803 V=800.0 PL=0
MOVL C01804 V=800.0 PL=0
MOVL C01805 V=800.0 PL=0
MOVL C01806 V=800.0 PL=0
MOVL C01807 V=800.0 PL=0
MOVL C01808 V=800.0 PL=0
MOVL C01809 V=800.0 PL=0
MOVL C01810 V=800.0 PL=0
MOVL C01811 V=800.0 PL=0
MOVL C01812 V=800.0 PL=0
MOVL C01813 V=800.0 PL=0
MOVL C01814 V=800.0 PL=0
MOVL C01815 V=800.0 PL=0
MOVL C01816 V=800.0 PL=0
MOVL C01817 V=800.0 PL=0
MOVL C01818 V=800.0 PL=0
MOVL C01819 V=800.0 PL=0
MOVL C01820 V=800.0 PL=0
MOVL C01821 V=800.0 PL=0
MOVL C01822 V=800.0 PL=0
MOVL C01823 V=800.0 PL=0
MOVL C01824 V=800.0 PL=0
MOVL C01825 V=800.0 PL=0
MOVL C01826 V=800.0 PL=0
MOVL C01827 V=800.0 PL=0
MOVL C01828 V=800.0 PL=0
MOVL C01829 V=800.0 PL=0
MOVL C01830 V=800.0 PL=0
MOVL C01831 V=800.0 PL=0
MOVL C01832 V=800.0 PL=0
MOVL C01833 V=800.0 PL=0
MOVL C01834 V=800.0 PL=0
MOVL C01835 V=800.0 PL=0
MOVL C01836 V=800.0 PL=0
MOVL C01837 V=800.0 PL=0
MOVL C01838 V=800.0 PL=0
MOVL C01839 V=800.0 PL=0
MOVL C01840 V=800.0 PL=0
MOVL C01841 V=800.0 PL=0
MOVL C01842 V=800.0 PL=0
MOVL C01843 V=800.0 PL=0
MOVL C01844 V=800.0 PL=0
MOVL C01845 V=800.0 PL=0
MOVL C01846 V=800.0 PL=0
MOVL C01847 V=800.0 PL=0
MOVL C01848 V=800.0 PL=0
MOVL C01849 V=800.0 PL=0
MOVL C01850 V=800.0 PL=0
MOVL C01851 V=800.0 PL=0
MOVL C01852 V=800.0 PL=0
MOVL C01853 V=800.0 PL=0
MOVL C01854 V=800.0 PL=0
MOVL C01855 V=800.0 PL=0
MOVL C01856 V=800.0 PL=0
MOVL C01857 V=800.0 PL=0
MOVL C01858 V=800.0 PL=0
MOVL C01859 V=800.0 PL=0
MOVL C01860 V=800.0 PL=0
MOVL C01861 V=800.0 PL=0
MOVL C01862 V=800.0 PL=0
MOVL C01863 V=800.0 PL=0
MOVL C01864 V=800.0 PL=0
MOVL C01865 V=800.0 PL=0
MOVL C01866 V=800.0 PL=0
MOVL C01867 V=800.0 PL=0
MOVL C01868 V=800.0 PL=0
MOVL C01869 V=800.0 PL=0
MOVL C01870 V=800.0 PL=0
MOVL C01871 V=800.0 PL=0
MOVL C01872 V=800.0 PL=0
MOVL C01873 V=800.0 PL=0
MOVL C01874 V=800.0 PL=0
MOVL C01875 V=800.0 PL=0
MOVL C01876 V=800.0 PL=0
MOVL C01877 V=800.0 PL=0
MOVL C01878 V=800.0 PL=0
MOVL C01879 V=800.0 PL=0
MOVL C01880 V=800.0 PL=0
MOVL C01881 V=800.0 PL=0
MOVL C01882 V=800.0 PL=0
MOVL C01883 V=800.0 PL=0
MOVL C01884 V=800.0 PL=0
MOVL C01885 V=800.0 PL=0
MOVL C01886 V=800.0 PL=0
MOVL C01887 V=800.0 PL=0
MOVL C01888 V=800.0 PL=0
MOVL C01889 V=800.0 PL=0
MOVL C01890 V=800.0 PL=0
MOVL C01891 V=800.0 PL=0
MOVL C01892 V=800.0 PL=0
MOVL C01893 V=800.0 PL=0
MOVL C01894 V=800.0 PL=0
MOVL C01895 V=800.0 PL=0
MOVL C01896 V=800.0 PL=0
MOVL C01897 V=800.0 PL=0
MOVL C01898 V=800.0 PL=0
MOVL C01899 V=800.0 PL=0
MOVL C01900 V=800.0 PL=0
MOVL C01901 V=800.0 PL=0
MOVL C01902 V=800.0 PL=0
MOVL C01903 V=800.0 PL=0
MOVL C01904 V=800.0 PL=0
MOVL C01905 V=800.0 PL=0
MOVL C01906 V=800.0 PL=0
MOVL C01907 V=800.0 PL=0
MOVL C01908 V=800.0 PL=0
MOVL C01909 V=800.0 PL=0
MOVL C01910 V=800.0 PL=0
MOVL C01911 V=800.0 PL=0
MOVL C01912 V=800.0 PL=0
MOVL C01913 V=800.0 PL=0
MOVL C01914 V=800.0 PL=0
MOVL C01915 V=800.0 PL=0
MOVL C01916 V=800.0 PL=0
MOVL C01917 V=800.0 PL=0
MOVL C01918 V=800.0 PL=0
MOVL C01919 V=800.0 PL=0
MOVL C01920 V=800.0 PL=0
MOVL C01921 V=800.0 PL=0
MOVL C01922 V=800.0 PL=0
MOVL C01923 V=800.0 PL=0
MOVL C01924 V=800.0 PL=0
MOVL C01925 V=800.0 PL=0
MOVL C01926 V=800.0 PL=0
MOVL C01927 V=800.0 PL=0
MOVL C01928 V=800.0 PL=0
MOVL C01929 V=800.0 PL=0
MOVL C01930 V=800.0 PL=0
MOVL C01931 V=800.0 PL=0
MOVL C01932 V=800.0 PL=0
MOVL C01933 V=800.0 PL=0
MOVL C01934 V=800.0 PL=0
MOVL C01935 V=800.0 PL=0
MOVL C01936 V=800.0 PL=0
MOVL C01937 V=800.0 PL=0
MOVL C01938 V=800.0 PL=0
MOVL C01939 V=800.0 PL=0
MOVL C01940 V=800.0 PL=0
MOVL C01941 V=800.0 PL=0
MOVL C01942 V=800.0 PL=0
MOVL C01943 V=800.0 PL=0
MOVL C01944 V=800.0 PL=0
MOVL C01945 V=800.0 PL=0
MOVL C01946 V=800.0 PL=0
MOVL C01947 V=800.0 PL=0
MOVL C01948 V=800.0 PL=0
MOVL C01949 V=800.0 PL=0
MOVL C01950 V=800.0 PL=0
MOVL C01951 V=800.0 PL=0
MOVL C01952 V=800.0 PL=0
MOVL C01953 V=800.0 PL=0
MOVL C01954 V=800.0 PL=0
MOVL C01955 V=800.0 PL=0
MOVL C01956 V=800.0 PL=0
MOVL C01957 V=800.0 PL=0
MOVL C01958 V=800.0 PL=0
MOVL C01959 V=800.0 PL=0
MOVL C01960 V=800.0 PL=0
MOVL C01961 V=800.0 PL=0
MOVL C01962 V=800.0 PL=0
MOVL C01963 V=800.0 PL=0
MOVL C01964 V=800.0 PL=0
MOVL C01965 V=800.0 PL=0
MOVL C01966 V=800.0 PL=0
MOVL C01967 V=800.0 PL=0
MOVL C01968 V=800.0 PL=0
MOVL C01969 V=800.0 PL=0
MOVL C01970 V=800.0 PL=0
MOVL C01971 V=800.0 PL=0
MOVL C01972 V=800.0 PL=0
MOVL C01973 V=800.0 PL=0
MOVL C01974 V=800.0 PL=0
MOVL C01975 V=800.0 PL=0
MOVL C01976 V=800.0 PL=0
MOVL C01977 V=800.0 PL=0
MOVL C01978 V=800.0 PL=0
MOVL C01979 V=800.0 PL=0
MOVL C01980 V=800.0 PL=0
MOVL C01981 V=800.0 PL=0
MOVL C01982 V=800.0 PL=0
MOVL C01983 V=800.0 PL=0
MOVL C01984 V=800.0 PL=0
MOVL C01985 V=800.0 PL=0
MOVL C01986 V=800.0 PL=0
MOVL C01987 V=800.0 PL=0
MOVL C01988 V=800.0 PL=0
MOVL C01989 V=800.0 PL=0
MOVL C01990 V=800.0 PL=0
MOVL C01991 V=800.0 PL=0
MOVL C01992 V=800.0 PL=0
MOVL C01993 V=800.0 PL=0
MOVL C01994 V=800.0 PL=0
MOVL C01995 V=800.0 PL=0
MOVL C01996 V=800.0 PL=0
MOVL C01997 V=800.0 PL=0
MOVL C01998 V=800.0 PL=0
MOVL C01999 V=800.0 PL=0
MOVL C02000 V=800.0 PL=0
MOVL C02001 V=800.0 PL=0
MOVL C02002 V=800.0 PL=0
MOVL C02003 V=800.0 PL=0
MOVL C02004 V=800.0 PL=0
MOVL C02005 V=800.0 PL=0
MOVL C02006 V=800.0 PL=0
MOVL C02007 V=800.0 PL=0
MOVL C02008 V=800.0 PL=0
MOVL C02009 V=800.0 PL=0
MOVL C02010 V=800.0 PL=0
MOVL C02011 V=800.0 PL=0
MOVL C02012 V=800.0 PL=0
MOVL C02013 V=800.0 PL=0
MOVL C02014 V=800.0 PL=0
MOVL C02015 V=800.0 PL=0
MOVL C02016 V=800.0 PL=0
MOVL C02017 V=800.0 PL=0
MOVL C02018 V=800.0 PL=0
MOVL C02019 V=800.0 PL=0
MOVL C02020 V=800.0 PL=0
MOVL C02021 V=800.0 PL=0
MOVL C02022 V=800.0 PL=0
MOVL C02023 V=800.0 PL=0
MOVL C02024 V=800.0 PL=0
MOVL C02025 V=800.0 PL=0
MOVL C02026 V=800.0 PL=0
MOVL C02027 V=800.0 PL=0
MOVL C02028 V=800.0 PL=0
MOVL C02029 V=800.0 PL=0
MOVL C02030 V=800.0 PL=0
MOVL C02031 V=800.0 PL=0
MOVL C02032 V=800.0 PL=0
MOVL C02033 V=800.0 PL=0
MOVL C02034 V=800.0 PL=0
MOVL C02035 V=800.0 PL=0
MOVL C02036 V=800.0 PL=0
MOVL C02037 V=800.0 PL=0
MOVL C02038 V=800.0 PL=0
MOVL C02039 V=800.0 PL=0
MOVL C02040 V=800.0 PL=0
MOVL C02041 V=800.0 PL=0
MOVL C02042 V=800.0 PL=0
MOVL C02043 V=800.0 PL=0
MOVL C02044 V=800.0 PL=0
MOVL C02045 V=800.0 PL=0
MOVL C02046 V=800.0 PL=0
MOVL C02047 V=800.0 PL=0
MOVL C02048 V=800.0 PL=0
MOVL C02049 V=800.0 PL=0
MOVL C02050 V=800.0 PL=0
MOVL C02051 V=800.0 PL=0
MOVL C02052 V=800.0 PL=0
MOVL C02053 V=800.0 PL=0
MOVL C02054 V=800.0 PL=0
MOVL C02055 V=800.0 PL=0
MOVL C02056 V=800.0 PL=0
MOVL C02057 V=800.0 PL=0
MOVL C02058 V=800.0 PL=0
MOVL C02059 V=800.0 PL=0
MOVL C02060 V=800.0 PL=0
MOVL C02061 V=800.0 PL=0
MOVL C02062 V=800.0 PL=0
MOVL C02063 V=800.0 PL=0
MOVL C02064 V=800.0 PL=0
MOVL C02065 V=800.0 PL=0
MOVL C02066 V=800.0 PL=0
MOVL C02067 V=800.0 PL=0
MOVL C02068 V=800.0 PL=0
MOVL C02069 V=800.0 PL=0
MOVL C02070 V=800.0 PL=0
MOVL C02071 V=800.0 PL=0
MOVL C02072 V=800.0 PL=0
MOVL C02073 V=800.0 PL=0
MOVL C02074 V=800.0 PL=0
MOVL C02075 V=800.0 PL=0
MOVL C02076 V=800.0 PL=0
MOVL C02077 V=800.0 PL=0
MOVL C02078 V=800.0 PL=0
MOVL C02079 V=800.0 PL=0
MOVL C02080 V=800.0 PL=0
MOVL C02081 V=800.0 PL=0
MOVL C02082 V=800.0 PL=0
MOVL C02083 V=800.0 PL=0
MOVL C02084 V=800.0 PL=0
MOVL C02085 V=800.0 PL=0
MOVL C02086 V=800.0 PL=0
MOVL C02087 V=800.0 PL=0
MOVL C02088 V=800.0 PL=0
MOVL C02089 V=800.0 PL=0
MOVL C02090 V=800.0 PL=0
MOVL C02091 V=800.0 PL=0
MOVL C02092 V=800.0 PL=0
MOVL C02093 V=800.0 PL=0
MOVL C02094 V=800.0 PL=0
MOVL C02095 V=800.0 PL=0
MOVL C02096 V=800.0 PL=0
MOVL C02097 V=800.0 PL=0
MOVL C02098 V=800.0 PL=0
MOVL C02099 V=800.0 PL=0
MOVL C02100 V=800.0 PL=0
MOVL C02101 V=800.0 PL=0
MOVL C02102 V=800.0 PL=0
MOVL C02103 V=800.0 PL=0
MOVL C02104 V=800.0 PL=0
MOVL C02105 V=800.0 PL=0
MOVL C02106 V=800.0 PL=0
MOVL C02107 V=800.0 PL=0
MOVL C02108 V=800.0 PL=0
MOVL C02109 V=800.0 PL=0
MOVL C02110 V=800.0 PL=0
MOVL C02111 V=800.0 PL=0
MOVL C02112 V=800.0 PL=0
MOVL C02113 V=800.0 PL=0
MOVL C02114 V=800.0 PL=0
MOVL C02115 V=800.0 PL=0
MOVL C02116 V=800.0 PL=0
MOVL C02117 V=800.0 PL=0
MOVL C02118 V=800.0 PL=0
MOVL C02119 V=800.0 PL=0
MOVL C02120 V=800.0 PL=0
MOVL C02121 V=800.0 PL=0
MOVL C02122 V=800.0 PL=0
MOVL C02123 V=800.0 PL=0
MOVL C02124 V=800.0 PL=0
MOVL C02125 V=800.0 PL=0
MOVL C02126 V=800.0 PL=0
MOVL C02127 V=800.0 PL=0
MOVL C02128 V=800.0 PL=0
MOVL C02129 V=800.0 PL=0
MOVL C02130 V=800.0 PL=0
MOVL C02131 V=800.0 PL=0
MOVL C02132 V=800.0 PL=0
MOVL C02133 V=800.0 PL=0
